# B&R Automation Studio project acopos6d_issues (part 4)

#### PackMLModuleStateManaging.cpp
```cpp
#include "PackMLModule.hpp"

		// -----------------------------------------------------------------------------

const char *internalInfoStateNames[] = { "Undefined",
	"Clearing",
	"Stopped",
	"Starting",
	"Idle",
	"Suspended",
	"Execute",
	"Stopping",
	"Aborting",
	"Aborted",
	"Holding",
	"Held",
	"Unholding",
	"Suspending",
	"Unsuspending",
	"Resetting",
	"Completing",
	"Completed",
	"",
	"",
	"",
	"",
	"",
	"",
	"",
	"",
	"",
	"",
	"",
	"",
	"Deactivating",
	"Deactivated",
	"Activating" };

const char *internalInfoModeNames[] = { "Undefined",
	"Production",
	"Maintenance",
	"Manual",
	""};

		// -----------------------------------------------------------------------------
		// we need to add complete cmd to the pattern
const unsigned long CMD_VALID_BIT_PATTERN_LIST[]
	= { 0,          0x00000080, 0x20004080, 0x000000C0, 0x000000C4, 0x0000A2C0,
	0x000092C0, 0x00000080, 0,          0x20000001, 0x000000C0, 0x000088C0,
	0x000000C0, 0x000000C0, 0x000000C0, 0x000000C0, 0x000000C0, 0x000040C0,
	0,          0,          0,          0,          0,          0,
	0,          0,          0,          0,          0,          0,
	0,          0x80000000, 0 };

// -----------------------------------------------------------------------------

PackMLModule* PackMLModule::getParentPtr(){
	if (!hasParent_)
		return nullptr;

	return pParentLink_;
}
// -----------------------------------------------------------------------------
PackMLModule* PackMLModule::getChildPtr(unsigned long int childIdx){
	if(childCount_ <= 0)
		return nullptr;

	return childLinks_[childIdx % childCount_];
}
// -----------------------------------------------------------------------------
PackMLModule* PackMLModule::getSiblingPtr(unsigned long int siblingIdx){
	if (!hasParent_)
		return nullptr;

	return pParentLink_->getChildPtr(siblingIdx);
}
// -----------------------------------------------------------------------------

PackMLModuleStateEnu PackMLModule::getChildCurrentState(unsigned long int childIndex){
	if(childCount_ <= 0)
		return ST_UNDEFINED;

	return childLinks_[childIndex % childCount_]->getCurrentState();
}
		// -----------------------------------------------------------------------------
long int PackMLModule::getChildCurrentSubState(unsigned long int childIndex){
	if(childCount_ <= 0)
		return 0;

	return childLinks_[childIndex % childCount_]->getCurrentSubState();
}
		// -----------------------------------------------------------------------------
bool PackMLModule::getChildStateComplete(unsigned long int childIndex){
	if(childCount_ <= 0)
		return false;

	return childLinks_[childIndex % childCount_]->getStateComplete();
}
		// -----------------------------------------------------------------------------
const char* PackMLModule::getChildName(unsigned long int childIndex){
	if(childCount_ <= 0)
		return "";

	return childLinks_[childIndex % childCount_]->getModuleName();
}
		// -----------------------------------------------------------------------------
PackMLModuleStateEnu PackMLModule::getSiblingCurrentState(unsigned long int siblingIndex){
	if (!hasParent_)
		return ST_UNDEFINED;

	return pParentLink_->getChildCurrentState(siblingIndex);
}
		// -----------------------------------------------------------------------------
long int PackMLModule::getSiblingCurrentSubState(unsigned long int siblingIndex){
	if (!hasParent_)
		return 0;

	return pParentLink_->getChildCurrentSubState(siblingIndex);
}
		// -----------------------------------------------------------------------------
bool PackMLModule::getSiblingStateComplete(unsigned long int siblingIndex){
	if (!hasParent_)
		return false;

	return pParentLink_->getChildStateComplete(siblingIndex);
}
		// -----------------------------------------------------------------------------
const char* PackMLModule::getSiblingName(unsigned long int siblingIndex){
	if (!hasParent_)
		return "";

	return pParentLink_->getChildName(siblingIndex);
}
		// -----------------------------------------------------------------------------
bool PackMLModule::isChild_(PackMLModule* pModule){
	for (unsigned short i = 0; i < childCount_; ++i) {
		if (childLinks_[i] == pModule) {
			return true;
		}
	}
	return false;
}
		// -----------------------------------------------------------------------------
unsigned long PackMLModule::getSiblingCount(){
	if (!hasParent_) {
		return 1;
	}
	return pParentLink_->getChildCount();
}
		// -----------------------------------------------------------------------------
bool PackMLModule::getSiblingsStateComplete(){
	if (!hasParent_) {
		return stateComplete_;
	}
	return pParentLink_->getChildrenStateComplete();
}

		// -----------------------------------------------------------------------------
bool PackMLModule::getChildrenStateComplete(){
	for (unsigned short i = 0; i < childCount_; ++i) {
		if (!childLinks_[i]->getStateComplete()) {
			return false;
		}
	}
	return true;
}
		// -----------------------------------------------------------------------------
PackMLModuleStateEnu PackMLModule::getParentCurrentState()
{
	if (!hasParent_) {
		return ST_UNDEFINED;
	}
	return pParentLink_->getCurrentState();
}

		// -----------------------------------------------------------------------------

long int PackMLModule::getParentCurrentSubState()
{
	if (!hasParent_) {
		return 0;
	}
	return pParentLink_->getCurrentSubState();
}

		// -----------------------------------------------------------------------------

const char *PackMLModule::getParentName()
{
	if (!hasParent_) {
		return "";
	}
	return pParentLink_->getModuleName();
}

bool PackMLModule::getParentStateComplete()
{
	if (!hasParent_) {
		return true;
	}
	return pParentLink_->getStateComplete();
}

		// -----------------------------------------------------------------------------

const char *PackMLModule::getCurrentStateStr() const
{
	return internalInfoStateNames[stateCurrent_];

}

const char *PackMLModule::getStateStr(PackMLModuleStateEnu state) const
{
	return internalInfoStateNames[state];
}

		// -----------------------------------------------------------------------------

		// -----------------------------------------------------------------------------

const char* PackMLModule::getCurrentModeName() const
{
	return internalInfoModeNames[modeCurrent_];
}

const char* PackMLModule::getModeName(signed long int modeId) const
{
	return internalInfoModeNames[modeId];
}

		// -----------------------------------------------------------------------------

// --------------------------------------------------------------------------

void PackMLModule::setNewModeCurrent(long int mode)
{
	modeCurrent_ = mode;

	for (unsigned short i = 0; i < childCount_; ++i) {
		childLinks_[i]->setNewModeCurrent(modeCurrent_);
	}
}

		// -----------------------------------------------------------------------------

bool PackMLModule::setCurrentMode(long int mode)
{

	// Check if the hierarchy is in synch
	if(!isModeChangePossible())
		return false;

	// update mode
	setNewModeCurrent(mode);
	// propagate mode to the children within one cycle
	return true;
}

		// -----------------------------------------------------------------------------

bool PackMLModule::isModeChangePossible()
{
	// What should the child do when it is not synchronised with the parent?
	if (!childrenInState_(stateCurrent_)) {
		return false;
	}

	for (unsigned short i = 0; i < childCount_; ++i) {
		if (!childLinks_[i]->isModeChangePossible()) {
			return false;
		}
	}

	return true;
}
		// -----------------------------------------------------------------------------

bool PackMLModule::childrenInState_(PackMLModuleStateEnu state)
{

	for (unsigned short i = 0; i < childCount_; ++i) {
		PackMLModuleStateEnu childState = childLinks_[i]->getCurrentState();
		if (childState != state && childState != ST_DEACTIVATED) {
			return false;
		}
	}
	return true;
}

		// -------------------------------------------------------------------------

bool PackMLModule::stateExistInPattern_(unsigned long stateBitPattern,
	PackMLModuleStateEnu state)
{
	if (state == ST_UNDEFINED) {
		return true;
	}
	unsigned long patternChecker = 1;
	return (stateBitPattern & (patternChecker << (state - 1)));
}

		// -------------------------------------------------------------------------

bool PackMLModule::cmdValid_(PackMLModuleStateEnu state)
{

	return stateExistInPattern_(CMD_VALID_BIT_PATTERN_LIST[stateCurrent_],
		state);
}

		// ------------------------------------------------------------------------

bool PackMLModule::isActingState(PackMLModuleStateEnu state)
{
	unsigned long actingStateBitPattern = 0xA000FAC5;

	return stateExistInPattern_(actingStateBitPattern, state);
}

		// -----------------------------------------------------------------------------

// from waiting state to acting state
void PackMLModule::executeCmd_(PackMLModuleStateEnu targetState)
{
	stateCurrent_ = targetState;
	// reset internal bools
	resetInternalCmds_();
	resetWaitingFor_();
	resetInteruptedBy_();
}

		// -----------------------------------------------------------------------------
// from acting state to waiting state
void PackMLModule::executeActingState_(PackMLModuleStateEnu targetState)
{
	if (childrenInSynch_(targetState)) {
		// Update the state
		stateCurrent_ = targetState;
		// reset internal bools
		resetInternalCmds_();
		resetWaitingFor_();
	}
}

		// -----------------------------------------------------------------------------
		// Checks if the children are in the desired state in case where they want to be
		// synchronised
bool PackMLModule::childrenInSynch_(PackMLModuleStateEnu targetState)
{

	for (unsigned long i = 0; i < childCount_; ++i) {
		if ((childLinks_[i]->getCurrentState() != targetState) && childLinks_[i]->needParentSynch(stateCurrent_)) {
			return false;
		}
	}
	return true;
}

		// -----------------------------------------------------------------------------

void PackMLModule::resetInternalCmds_()
{
	if(isActingState(stateCurrent_)){
		externalAbort_ = false;
		externalClear_ = false;
		externalStop_ = false;
		externalReset_ = false;
		externalStart_ = false;
		externalHold_ = false;
		externalUnhold_ = false;
		externalSuspend_ = false;
		externalUnsuspend_ = false;
		externalComplete_ = false;
		externalStateComplete_ = false;
	}

	activate_ = false;
	deactivate_ = false;

	abort_ = externalAbort_;
	clear_ = externalClear_;
	stop_ = externalStop_;
	reset_ = externalReset_;
	start_ = externalStart_;
	hold_ = externalHold_;
	unhold_ = externalUnhold_;
	suspend_ = externalSuspend_;
	unsuspend_ = externalUnsuspend_;
	complete_ = externalComplete_;
	stateComplete_ = false;

	oldAbort_ = false;
	oldClear_ = false;
	oldStop_ = false;
	oldReset_ = false;
	oldStart_ = false;
	oldHold_ = false;
	oldUnhold_ = false;
	oldSuspend_ = false;
	oldUnsuspend_ = false;
	oldComplete_ = false;
	oldStateComplete_ = false;

	timeInState_ = 0.0;
}

		// -----------------------------------------------------------------------------

void PackMLModule::escalateCmdAbort()
{
	if (escalateAbort_) {
		return pParentLink_->escalateCmdAbort();
	}
	abort_ = !overrideAbort_;
	externalAbort_ = abort_;
}
void PackMLModule::escalateCmdClear()
{
	if (escalateClear_) {
		return pParentLink_->escalateCmdClear();
	}
	clear_ = !overrideClear_;
	externalClear_ = clear_;
}
void PackMLModule::escalateCmdStop()
{
	if (escalateStop_) {
		return pParentLink_->escalateCmdStop();
	}
	stop_ = !overrideStop_;
	externalStop_ = stop_;
}
void PackMLModule::escalateCmdReset()
{
	if (escalateReset_) {
		return pParentLink_->escalateCmdReset();
	}
	reset_ = !overrideReset_;
	externalReset_ = reset_;
}
void PackMLModule::escalateCmdHold()
{
	if (escalateHold_) {
		return pParentLink_->escalateCmdHold();
	}
	hold_ = !overrideHold_;
	externalHold_ = hold_;
}
void PackMLModule::escalateCmdUnhold()
{
	if (escalateUnhold_) {
		return pParentLink_->escalateCmdUnhold();
	}
	unhold_ = !overrideUnhold_;
	externalUnhold_ = unhold_;
}
void PackMLModule::escalateCmdSuspend()
{
	if (escalateSuspend_) {
		return pParentLink_->escalateCmdSuspend();
	}
	suspend_ = !overrideSuspend_;
	externalSuspend_ = suspend_;
}
void PackMLModule::escalateCmdUnsuspend()
{
	if (escalateUnsuspend_) {
		return pParentLink_->escalateCmdUnsuspend();
	}
	unsuspend_ = !overrideUnsuspend_;
	externalUnsuspend_ = unsuspend_;
}
void PackMLModule::escalateCmdStart()
{
	if (escalateStart_) {
		return pParentLink_->escalateCmdStart();
	}
	start_ = !overrideStart_;
	externalStart_ = start_;
}
void PackMLModule::escalateCmdComplete()
{
	if (escalateComplete_) {
		return pParentLink_->escalateCmdComplete();
	}
	complete_ = !overrideComplete_;
	externalComplete_ = complete_;
}

// ----------------------------------------------------------------------------

void PackMLModule::propagateCmdAbort(bool root)
{
	abort_ = reactToAbort_ && !root;
	externalAbort_ = abort_;

	for (unsigned short i = 0; i < childCount_; ++i) {
		childLinks_[i]->propagateCmdAbort(false);
	}
}
void PackMLModule::propagateCmdClear(bool root)
{
	clear_ = reactToClear_ && !root;
	externalClear_ = clear_;

	for (unsigned short i = 0; i < childCount_; ++i) {
		childLinks_[i]->propagateCmdClear(false);
	}
}
void PackMLModule::propagateCmdStop(bool root)
{
	stop_ = reactToStop_ && !root;
	externalStop_ = stop_;

	for (unsigned short i = 0; i < childCount_; ++i) {
		childLinks_[i]->propagateCmdStop(false);
	}
}
void PackMLModule::propagateCmdReset(bool root)
{
	reset_ = reactToReset_ && !root;
	externalReset_ = reset_;

	for (unsigned short i = 0; i < childCount_; ++i) {
		childLinks_[i]->propagateCmdReset(false);
	}
}
void PackMLModule::propagateCmdHold(bool root)
{
	hold_ = reactToHold_ && !root;
	externalHold_ = hold_;

	for (unsigned short i = 0; i < childCount_; ++i) {
		childLinks_[i]->propagateCmdHold(false);
	}
}
void PackMLModule::propagateCmdUnhold(bool root)
{
	unhold_ = reactToUnhold_ && !root;
	externalUnhold_ = unhold_;

	for (unsigned short i = 0; i < childCount_; ++i) {
		childLinks_[i]->propagateCmdUnhold(false);
	}
}
void PackMLModule::propagateCmdSuspend(bool root)
{
	suspend_ = reactToSuspend_ && !root;
	externalSuspend_ = suspend_;

	for (unsigned short i = 0; i < childCount_; ++i) {
		childLinks_[i]->propagateCmdSuspend(false);
	}
}
void PackMLModule::propagateCmdUnsuspend(bool root)
{
	unsuspend_ = reactToUnsuspend_ && !root;
	externalUnsuspend_ = unsuspend_;

	for (unsigned short i = 0; i < childCount_; ++i) {
		childLinks_[i]->propagateCmdUnsuspend(false);
	}
}
void PackMLModule::propagateCmdStart(bool root)
{
	start_ = reactToStart_ && !root;
	externalStart_ = start_;

	for (unsigned short i = 0; i < childCount_; ++i) {
		childLinks_[i]->propagateCmdStart(false);
	}
}
void PackMLModule::propagateCmdComplete(bool root)
{
	complete_ = reactToComplete_ && !root;
	externalComplete_ = complete_;

	for (unsigned short i = 0; i < childCount_; ++i) {
		childLinks_[i]->propagateCmdComplete(false);
	}
}

// ----------------------------------------------------------------------------

bool PackMLModule::evaluateCmdAbort(bool& newCmd)
{
	if (newCmd && !oldAbort_) {
		oldAbort_ = true;
		return setCmd_(ST_ABORTING);
	}
	else if (!newCmd && oldAbort_) {
		oldAbort_ = false;
		resetCmd_(ST_ABORTING);
	}
	return true;
}
bool PackMLModule::evaluateCmdStop(bool& newCmd)
{
	if (newCmd && !oldStop_) {
		oldStop_ = true;
		return setCmd_(ST_STOPPING);
	}
	else if (!newCmd && oldStop_) {
		oldStop_ = false;
		resetCmd_(ST_STOPPING);
	}
	return true;
}
bool PackMLModule::evaluateCmdClear(bool& newCmd)
{
	if (newCmd && !oldClear_) {
		oldClear_ = true;
		return setCmd_(ST_CLEARING);
	}
	else if (!newCmd && oldClear_) {
		oldClear_ = false;
		resetCmd_(ST_CLEARING);
	}
	return true;
}
bool PackMLModule::evaluateCmdReset(bool& newCmd)
{
	if (newCmd && !oldReset_) {
		oldReset_ = true;
		return setCmd_(ST_RESETTING);
	}
	else if (!newCmd && oldReset_) {
		oldReset_ = false;
		resetCmd_(ST_RESETTING);
	}
	return true;
}
bool PackMLModule::evaluateCmdStart(bool& newCmd)
{
	if (newCmd && !oldStart_) {
		oldStart_ = true;
		return setCmd_(ST_STARTING);
	}
	else if (!newCmd && oldStart_) {
		oldStart_ = false;
		resetCmd_(ST_STARTING);
	}
	return true;
}
bool PackMLModule::evaluateCmdSuspend(bool& newCmd)
{
	if (newCmd && !oldSuspend_) {
		oldSuspend_ = true;
		return setCmd_(ST_SUSPENDING);
	}
	else if (!newCmd && oldSuspend_) {
		oldSuspend_ = false;
		resetCmd_(ST_SUSPENDING);
	}
	return true;
}
bool PackMLModule::evaluateCmdUnsuspend(bool& newCmd)
{
	if (newCmd && !oldUnsuspend_) {
		oldUnsuspend_ = true;
		return setCmd_(ST_UNSUSPENDING);
	}
	else if (!newCmd && oldUnsuspend_) {
		oldUnsuspend_ = false;
		resetCmd_(ST_UNSUSPENDING);
	}
	return true;
}
bool PackMLModule::evaluateCmdHold(bool& newCmd)
{
	if (newCmd && !oldHold_) {
		oldHold_ = true;
		return setCmd_(ST_HOLDING);
	}
	else if (!newCmd && oldHold_) {
		oldHold_ = false;
		resetCmd_(ST_HOLDING);
	}
	return true;
}
bool PackMLModule::evaluateCmdUnhold(bool& newCmd)
{
	if (newCmd && !oldUnhold_) {
		oldUnhold_ = true;
		return setCmd_(ST_UNHOLDING);
	}
	else if (!newCmd && oldUnhold_) {
		oldUnhold_ = false;
		resetCmd_(ST_UNHOLDING);
	}
	return true;
}
bool PackMLModule::evaluateCmdComplete(bool& newCmd)
{
	if (newCmd && !oldComplete_) {
		oldComplete_ = true;
		return setCmd_(ST_COMPLETING);
	}
	else if (!newCmd && oldComplete_) {
		oldComplete_ = false;
		resetCmd_(ST_COMPLETING);
	}
	return true;
}
bool PackMLModule::evaluateCmdStateComplete(bool& newCmd)
{
	if (newCmd && !oldStateComplete_) {
		oldStateComplete_ = true;
		return setCmd_(ST_UNDEFINED);
	}
	else if (!newCmd && oldStateComplete_) {
		oldStateComplete_ = false;
		resetCmd_(ST_UNDEFINED);
	}
	return true;
}

bool PackMLModule::setCmdAbort(){
	return setCmd_(ST_ABORTING);
}
bool PackMLModule::setCmdStop(){
	return setCmd_(ST_STOPPING);
}
bool PackMLModule::setCmdClear(){
	return setCmd_(ST_CLEARING);
}
bool PackMLModule::setCmdReset(){
	return setCmd_(ST_RESETTING);
}
bool PackMLModule::setCmdStart(){
	return setCmd_(ST_STARTING);
}
bool PackMLModule::setCmdSuspend(){
	return setCmd_(ST_SUSPENDING);
}
bool PackMLModule::setCmdUnsuspend(){
	return setCmd_(ST_UNSUSPENDING);
}
bool PackMLModule::setCmdHold(){
	return setCmd_(ST_HOLDING);
}
bool PackMLModule::setCmdUnhold(){
	return setCmd_(ST_UNHOLDING);
}
bool PackMLModule::setCmdComplete(){
	return setCmd_(ST_COMPLETING);
}
bool PackMLModule::setCmdStateComplete(){
	return setCmd_(ST_UNDEFINED);
}

void PackMLModule::resetCmdAbort(){
	return resetCmd_(ST_ABORTING);
}
void PackMLModule::resetCmdStop(){
	return resetCmd_(ST_STOPPING);
}
void PackMLModule::resetCmdClear(){
	return resetCmd_(ST_CLEARING);
}
void PackMLModule::resetCmdReset(){
	return resetCmd_(ST_RESETTING);
}
void PackMLModule::resetCmdStart(){
	return resetCmd_(ST_STARTING);
}
void PackMLModule::resetCmdSuspend(){
	return resetCmd_(ST_SUSPENDING);
}
void PackMLModule::resetCmdUnsuspend(){
	return resetCmd_(ST_UNSUSPENDING);
}
void PackMLModule::resetCmdHold(){
	return resetCmd_(ST_HOLDING);
}
void PackMLModule::resetCmdUnhold(){
	return resetCmd_(ST_UNHOLDING);
}
void PackMLModule::resetCmdComplete(){
	return resetCmd_(ST_COMPLETING);
}
void PackMLModule::resetCmdStateComplete(){
	return resetCmd_(ST_UNDEFINED);
}

		// -----------------------------------------------------------------------------

bool PackMLModule::setCmd_(PackMLModuleStateEnu targetActingState) // NOLINT
{

	bool cmdValid = cmdValid_(targetActingState);

	switch (targetActingState) { // NOCCM
		case ST_CLEARING:
			if (overrideClear_ && !escalateClear_) {
				return false; // error code
			}
			if (hasParent_ && escalateClear_ && cmdValid) {
				pParentLink_->escalateCmdClear();
				setInteruptedBy_();
			}
			clear_ = !overrideClear_; //!overrideAbort_ || !escalateAbort_;
			break;

		case ST_STARTING:
			if (overrideStart_ && !escalateStart_) {
				return false; // error code
			}
			if (hasParent_ && escalateStart_ && cmdValid) {
				pParentLink_->escalateCmdStart();
				setInteruptedBy_();
			}
			start_ = !overrideStart_;
			break;

		case ST_STOPPING:
			if (overrideStop_ && !escalateStop_) {
				return false; // error code
			}
			if (hasParent_ && escalateStop_) {
				pParentLink_->escalateCmdStop();
			}
			if(cmdValid){
				setInteruptedBy_();
				stop_ = !overrideStop_;
			}
			break;

		case ST_ABORTING:
			if (overrideAbort_ && !escalateAbort_) {
				return false; // error code
			}
			if (hasParent_ && escalateAbort_) {
				pParentLink_->escalateCmdAbort();
			}

			if(cmdValid){
				setInteruptedBy_();
				abort_ = !overrideAbort_;
			}
			break;

		case ST_HOLDING:
			if (overrideHold_ && !escalateHold_) {
				return false; // error code
			}
			if (hasParent_ && escalateHold_) {
				pParentLink_->escalateCmdHold();
			}
			if(cmdValid){
				setInteruptedBy_();
				hold_ = !overrideHold_;
			}
			break;

		case ST_UNHOLDING:
			if (overrideUnhold_ && !escalateUnhold_) {
				return false; // error code
			}
			if (hasParent_ && escalateUnhold_ && cmdValid) {
				pParentLink_->escalateCmdUnhold();
				setInteruptedBy_();
			}
			unhold_ = !overrideUnhold_;
			break;

		case ST_SUSPENDING:
			if (overrideSuspend_ && !escalateSuspend_) {
				return false; // error code
			}
			if (hasParent_ && escalateSuspend_) {
				pParentLink_->escalateCmdSuspend();
			}
			if(cmdValid){
				setInteruptedBy_();
				suspend_ = !overrideSuspend_;
			}
			break;

		case ST_UNSUSPENDING:
			if (overrideUnsuspend_ && !escalateUnsuspend_) {
				return false; // error code
			}
			if (hasParent_ && escalateUnsuspend_ && cmdValid) {
				pParentLink_->escalateCmdUnsuspend();
				setInteruptedBy_();
			}
			unsuspend_ = !overrideUnsuspend_;
			break;

		case ST_RESETTING:
			if (overrideReset_ && !escalateReset_) {
				return false; // error code
			}
			if (hasParent_ && escalateReset_ && cmdValid) {
				pParentLink_->escalateCmdReset();
				setInteruptedBy_();
			}
			reset_ = !overrideReset_;
			break;

		case ST_COMPLETING:
			// check if the state group is configured
			if (overrideComplete_ && !escalateComplete_) {
				return false; // error code
			}
			if (hasParent_ && escalateComplete_) {
				pParentLink_->escalateCmdComplete();
			}
			if(cmdValid){
				setInteruptedBy_();
				complete_ = !overrideComplete_;
			}
			break;

		case ST_UNDEFINED:
			stateComplete_ = true;
			break;

		default:
			break;
	}

	return true;
}

		// -----------------------------------------------------------------------------

void PackMLModule::resetCmd_(PackMLModuleStateEnu targetActingState)
{

	switch (targetActingState) { // NOCCM
		case ST_CLEARING:
			clear_ = externalClear_;
			break;

		case ST_STARTING:
			start_ = externalStart_;
			break;

		case ST_STOPPING:
			stop_ = externalStop_;
			break;

		case ST_ABORTING:
			abort_ = externalAbort_;
			break;

		case ST_HOLDING:
			hold_ = externalHold_;
			break;

		case ST_UNHOLDING:
			unhold_ = externalUnhold_;
			break;

		case ST_SUSPENDING:
			suspend_ = externalSuspend_;
			break;

		case ST_UNSUSPENDING:
			unsuspend_ = externalUnsuspend_;
			break;

		case ST_RESETTING:
			reset_ = externalReset_;
			break;

		case ST_COMPLETING:
			complete_ = externalComplete_;
			break;

		case ST_UNDEFINED:
			stateComplete_ = externalStateComplete_;
			break;

		default:
			break;
	}
}

		// -----------------------------------------------------------------------------

		// if parent synchronisation needed
bool PackMLModule::needParentSynch(PackMLModuleStateEnu state)
{
	if (hierarchyLevel_ == 0) {
		return true;
	}

	switch (stateCurrent_) { // NOCCM

		case ST_CLEARING:
			switch (state) { // NOCCM
				case ST_ABORTING:
					return overrideAbort_ || reactToAbort_;
				case ST_CLEARING:
					return overrideClear_ || reactToClear_;
				default:
					break;
			}
			break;

		case ST_STOPPED:
			switch (state) { // NOCCM
				case ST_ABORTING:
					return overrideAbort_ || reactToAbort_;
				case ST_RESETTING:
					return overrideReset_ || reactToReset_;
				default:
					break;
			}
			break;

		case ST_IDLE:
			switch (state) { // NOCCM
				case ST_ABORTING:
					return overrideAbort_ || reactToAbort_;
				case ST_STOPPING:
					return overrideStop_ || reactToStop_;
				case ST_STARTING:
					return overrideStart_ || reactToStart_;
				default:
					break;
			}
			break;

		case ST_SUSPENDED:
			switch (state) { // NOCCM
				case ST_ABORTING:
					return overrideAbort_ || reactToAbort_;
				case ST_STOPPING:
					return overrideStop_ || reactToStop_;
				case ST_UNSUSPENDING:
					return overrideUnsuspend_ || reactToUnsuspend_;
				case ST_HOLDING:
					return overrideHold_ || reactToHold_;
				case ST_COMPLETING:
					return overrideComplete_ || reactToComplete_;
				default:
					break;
			}
			break;

		case ST_EXECUTE:
			switch (state) { // NOCCM
				case ST_ABORTING:
					return overrideAbort_ || reactToAbort_;
				case ST_STOPPING:
					return overrideStop_ || reactToStop_;
				case ST_SUSPENDING:
					return overrideSuspend_ || reactToSuspend_;
				case ST_HOLDING:
					return overrideHold_ || reactToHold_;
				case ST_COMPLETING:
					return overrideComplete_ || reactToComplete_;
				default:
					break;
			}
			break;

		case ST_STOPPING:
			switch (state) { // NOCCM
				case ST_ABORTING:
					return overrideAbort_ || reactToAbort_;
				case ST_STOPPING:
					return overrideStop_ || reactToStop_;
				default:
					break;
			}
			break;

		case ST_ABORTING:
			switch (state) { // NOCCM
				case ST_ABORTING:
					return overrideAbort_ || reactToAbort_;
				default:
					break;
			}
			break;

		case ST_ABORTED:
			switch (state) { // NOCCM
				case ST_CLEARING:
					return overrideClear_ || reactToClear_;
				default:
					break;
			}
			break;

		case ST_HELD:
			switch (state) { // NOCCM
				case ST_ABORTING:
					return overrideAbort_ || reactToAbort_;
				case ST_STOPPING:
					return overrideStop_ || reactToStop_;
				case ST_UNHOLDING:
					return overrideUnhold_ || reactToUnhold_;
				case ST_COMPLETING:
					return overrideComplete_ || reactToComplete_;
				default:
					break;
			}
			break;

		case ST_SUSPENDING:
			switch (state) { // NOCCM
				case ST_ABORTING:
					return overrideAbort_ || reactToAbort_;
				case ST_STOPPING:
					return overrideStop_ || reactToStop_;
				case ST_SUSPENDING:
					return overrideSuspend_ || reactToSuspend_;
				default:
					break;
			}
			break;
		case ST_UNSUSPENDING:
			switch (state) { // NOCCM
				case ST_ABORTING:
					return overrideAbort_ || reactToAbort_;
				case ST_STOPPING:
					return overrideStop_ || reactToStop_;
				case ST_UNSUSPENDING:
					return overrideUnsuspend_ || reactToUnsuspend_;
				default:
					break;
			}
			break;
		case ST_COMPLETING:
			switch (state) { // NOCCM
				case ST_ABORTING:
					return overrideAbort_ || reactToAbort_;
				case ST_STOPPING:
					return overrideStop_ || reactToStop_;
				case ST_COMPLETING:
					return overrideComplete_ || reactToComplete_;
				default:
					break;
			}
			break;
		case ST_STARTING:
			switch (state) { // NOCCM
				case ST_ABORTING:
					return overrideAbort_ || reactToAbort_;
				case ST_STOPPING:
					return overrideStop_ || reactToStop_;
				case ST_STARTING:
					return overrideStart_ || reactToStart_;
				default:
					break;
			}
			break;
		case ST_HOLDING:
			switch (state) { // NOCCM
				case ST_ABORTING:
					return overrideAbort_ || reactToAbort_;
				case ST_STOPPING:
					return overrideStop_ || reactToStop_;
				case ST_HOLDING:
					return overrideHold_ || reactToHold_;
				default:
					break;
			}
			break;
		case ST_UNHOLDING:
			switch (state) { // NOCCM
				case ST_ABORTING:
					return overrideAbort_ || reactToAbort_;
				case ST_STOPPING:
					return overrideStop_ || reactToStop_;
				case ST_UNHOLDING:
					return overrideUnhold_ || reactToUnhold_;
				default:
					break;
			}
			break;

		case ST_RESETTING:
			switch (state) { // NOCCM
				case ST_ABORTING:
					return overrideAbort_ || reactToAbort_;
				case ST_STOPPING:
					return overrideStop_ || reactToStop_;
				case ST_RESETTING:
					return overrideReset_ || reactToReset_;
				default:
					break;
			}
			break;

		case ST_COMPLETE:
			switch (state) { // NOCCM
				case ST_ABORTING:
					return overrideAbort_ || reactToAbort_;
				case ST_STOPPING:
					return overrideStop_ || reactToStop_;
				case ST_RESETTING:
					return overrideReset_ || reactToReset_;
				default:
					break;
			}
			break;

		default:
			break;
	}

	return false;
}

// -----------------------------------------------------------------------------
// decide if reacto to only should when parent + 1 state in front of child. e.g. instead of ST_ABORTING and ST_ABORTED --> only ST_ABORTING
void PackMLModule::checkParentStateCondition_()
{
	if (hierarchyLevel_ == 0) {
		return;
	}

	PackMLModuleStateEnu parentState = getParentCurrentState();

	if (parentState == stateCurrent_) {
		return;
	}

	switch (stateCurrent_) { // NOCCM
		case ST_CLEARING:
			switch (parentState) { // NOCCM
				case ST_ABORTING:
					abort_ = overrideAbort_ || abort_ || reactToAbort_;
					break;
				case ST_ABORTED:
					abort_ = overrideAbort_ || abort_;
					break;
				default:
					break;
			}
			break;

		case ST_STOPPED:
			switch (parentState) { // NOCCM
				case ST_ABORTING:
					abort_ = overrideAbort_ || abort_ || reactToAbort_;
					break;
				case ST_ABORTED:
					abort_ = overrideAbort_ || abort_;
					break;

				case ST_DEACTIVATING:
				case ST_DEACTIVATED:
					deactivate_ = (activationCondition_ == 1);
					break;

				case ST_RESETTING:
					reset_ = overrideReset_ || reset_ || reactToReset_;
					break;

				case ST_IDLE:
				case ST_STARTING:
				case ST_SUSPENDED:
				case ST_EXECUTE:
				case ST_HOLDING:
				case ST_HELD:
				case ST_UNHOLDING:
				case ST_SUSPENDING:
				case ST_UNSUSPENDING:
				case ST_COMPLETING:
				case ST_COMPLETE:
					reset_ = overrideReset_ || reset_;
					break;

				default:
					break;
			}
			break;

		case ST_IDLE:
			switch (parentState) { // NOCCM
				case ST_ABORTING:
					abort_ = overrideAbort_ || abort_ || reactToAbort_;
					break;
				case ST_ABORTED:
					abort_ = overrideAbort_ || abort_;
					break;

				case ST_CLEARING:
					stop_ = overrideStop_ || stop_;
					abort_ = (overrideAbort_ || abort_) && !stop_;
					break;

				case ST_STOPPING:
					stop_ = overrideStop_ || stop_ || reactToStop_;
					break;
				case ST_STOPPED:
					stop_ = overrideStop_ || stop_;
					break;

				case ST_DEACTIVATING:
				case ST_DEACTIVATED:
				case ST_ACTIVATING:
					stop_ = overrideStop_ || stop_;
					abort_ = (overrideAbort_ || abort_) && !stop_;
					break;

				case ST_STARTING:
					start_ = overrideStart_ || start_ || reactToStart_;
					break;

				case ST_EXECUTE:
				case ST_SUSPENDED:
				case ST_HOLDING:
				case ST_HELD:
				case ST_UNHOLDING:
				case ST_SUSPENDING:
				case ST_UNSUSPENDING:
				case ST_COMPLETING:
				case ST_COMPLETE:
					start_ = overrideStart_ || start_;
					break;

				default:
					break;
			}
			break;

		case ST_SUSPENDED:
			switch (parentState) { // NOCCM
				case ST_ABORTING:
					abort_ = overrideAbort_ || abort_ || reactToAbort_;
					break;
				case ST_ABORTED:
					abort_ = overrideAbort_ || abort_;
					break;

				case ST_CLEARING:
					stop_ = overrideStop_ || stop_;
					abort_ = (overrideAbort_ || abort_) && !stop_;
					break;

				case ST_STOPPING:
					stop_ = overrideStop_ || stop_ || reactToStop_;
					break;
				case ST_STOPPED:
					stop_ = overrideStop_ || stop_;
					break;

				case ST_UNSUSPENDING:
					unsuspend_ = overrideUnsuspend_ || unsuspend_ || reactToUnsuspend_;
					break;

				case ST_DEACTIVATING:
				case ST_DEACTIVATED:
				case ST_ACTIVATING:
					stop_ = overrideStop_ || stop_;
					abort_ = (overrideAbort_ || abort_) && !stop_;
					break;

				case ST_RESETTING:
				case ST_IDLE: // **********************
					unsuspend_ = overrideUnsuspend_ || unsuspend_;
					stop_ = (overrideStop_ || stop_) && !unsuspend_;
					break;

				case ST_COMPLETING:
					complete_ = overrideComplete_ || complete_ || reactToComplete_;
					break;
				case ST_COMPLETE:
					complete_ = overrideComplete_ || complete_;
					break;

				case ST_HOLDING:
					hold_ = overrideHold_ || hold_ || reactToHold_;
					break;
				case ST_HELD:
					hold_ = overrideHold_ || hold_;
					break;

				case ST_EXECUTE:
				case ST_STARTING:
				case ST_UNHOLDING:
					unsuspend_ = overrideUnsuspend_ || unsuspend_;
					break;

				default:
					break;
			}
			break;

		case ST_EXECUTE:
			switch (parentState) { // NOCCM
				case ST_ABORTING:
					abort_ = overrideAbort_ || abort_ || reactToAbort_;
					break;
				case ST_ABORTED:
					abort_ = overrideAbort_ || abort_;
					break;

				case ST_CLEARING:
					stop_ = overrideStop_ || stop_;
					abort_ = (overrideAbort_ || abort_) && !stop_;
					break;

				case ST_STOPPING:
					stop_ = overrideStop_ || stop_ || reactToStop_;
					break;

				case ST_STOPPED:
					stop_ = overrideStop_ || stop_;
					break;

				case ST_SUSPENDING:
					suspend_ = overrideSuspend_ || suspend_ || reactToSuspend_;
					break;

				case ST_SUSPENDED:
					suspend_ = overrideSuspend_ || suspend_;
					break;

				case ST_HOLDING:
					hold_ = overrideHold_ || hold_ || reactToHold_;
					break;

				case ST_HELD:
					hold_ = overrideHold_ || hold_;
					break;

				case ST_COMPLETING:
					complete_ = overrideComplete_ || complete_ || reactToComplete_;
					break;

				case ST_COMPLETE:
					complete_ = overrideComplete_ || complete_;
					break;

				case ST_DEACTIVATING:
				case ST_DEACTIVATED:
				case ST_ACTIVATING:
					stop_ = overrideStop_ || stop_;
					abort_ = (overrideAbort_ || abort_) && !stop_;
					break;

				case ST_RESETTING:
				case ST_IDLE:
					complete_ = overrideComplete_ || complete_;
					stop_ = (overrideStop_ || stop_) && !complete_;
					break;

				default:
					break;
			}
			break;

		case ST_STOPPING:
			switch (parentState) { // NOCCM
				case ST_ABORTING:
					abort_ = overrideAbort_ || abort_ || reactToAbort_;
					break;
				case ST_ABORTED:
					abort_ = overrideAbort_ || abort_;
					break;
				default:
					break;
			}
			break;

		case ST_ABORTED:
			switch (parentState) { // NOCCM
				case ST_DEACTIVATING:
				case ST_DEACTIVATED:
					deactivate_ = (activationCondition_ == 1);
					break;

				case ST_CLEARING:
					clear_ = overrideClear_ || clear_ || reactToClear_;
					break;

				case ST_STOPPED:
				case ST_STARTING:
				case ST_IDLE:
				case ST_SUSPENDED:
				case ST_EXECUTE:
				case ST_STOPPING:
				case ST_HOLDING:
				case ST_HELD:
				case ST_UNHOLDING:
				case ST_SUSPENDING:
				case ST_UNSUSPENDING:
				case ST_RESETTING:
				case ST_COMPLETING:
				case ST_COMPLETE:
				case ST_ACTIVATING:
					clear_ = overrideClear_ || clear_;
					break;

				default:
					break;
			}
			break;

		case ST_HELD:
			switch (parentState) { // NOCCM
				case ST_ABORTING:
					abort_ = overrideAbort_ || abort_ || reactToAbort_;
					break;
				case ST_ABORTED:
					abort_ = overrideAbort_ || abort_;
					break;

				case ST_CLEARING:
					stop_ = overrideStop_ || stop_;
					abort_ = (overrideAbort_ || abort_) && !stop_;
					break;

				case ST_STOPPING:
					stop_ = overrideStop_ || stop_ || reactToStop_;
					break;

				case ST_STOPPED:
					stop_ = overrideStop_ || stop_;
					break;

				case ST_UNHOLDING:
					unhold_ = overrideUnhold_ || unhold_ || reactToUnhold_;
					break;

				case ST_DEACTIVATING:
				case ST_DEACTIVATED:
				case ST_ACTIVATING:
					stop_ = overrideStop_ || stop_;
					abort_ = (overrideAbort_ || abort_) && !stop_;
					break;

				case ST_RESETTING:
				case ST_IDLE: // **********************
					unhold_ = overrideUnhold_ || unhold_;
					stop_ = (overrideStop_ || stop_) && !unhold_;
					break;

				case ST_COMPLETING:
					complete_ = overrideComplete_ || complete_ || reactToComplete_;
					break;
				case ST_COMPLETE:
					complete_ = overrideComplete_ || complete_;
					break;

				case ST_EXECUTE:
				case ST_SUSPENDING:
				case ST_SUSPENDED:
				case ST_UNSUSPENDING:
				case ST_STARTING:
					unhold_ = overrideUnhold_ || unhold_;
					break;

				default:
					break;
			}
			break;

		case ST_STARTING:
		case ST_HOLDING:
		case ST_UNHOLDING:
		case ST_SUSPENDING:
		case ST_UNSUSPENDING:
			switch (parentState) { // NOCCM
				case ST_ABORTING:
					abort_ = overrideAbort_ || abort_ || reactToAbort_;
					break;

				case ST_ABORTED:
					abort_ = overrideAbort_ || abort_;
					break;

				case ST_CLEARING:
					stop_ = overrideStop_ || stop_;
					abort_ = (overrideAbort_ || abort_) && !stop_;
					break;

				case ST_STOPPING:
					stop_ = overrideStop_ || stop_ || reactToStop_;
					break;

				case ST_STOPPED:
					stop_ = overrideStop_ || stop_;
					break;

				case ST_DEACTIVATING:
				case ST_DEACTIVATED:
				case ST_ACTIVATING:
					stop_ = overrideStop_ || stop_;
					abort_ = (overrideAbort_ || abort_) && !stop_;
					break;

				case ST_RESETTING:
				case ST_IDLE:
					stop_ = overrideStop_ || stop_;
					break;

				default:
					break;
			}
			break;

		case ST_RESETTING:
		case ST_COMPLETING:
			switch (parentState) { // NOCCM
				case ST_ABORTING:
					abort_ = overrideAbort_ || abort_ || reactToAbort_;
					break;
				case ST_ABORTED:
					abort_ = overrideAbort_ || abort_;
					break;

				case ST_CLEARING:
					stop_ = overrideStop_ || stop_;
					abort_ = (overrideAbort_ || abort_) && !stop_;
					break;

				case ST_STOPPING:
					stop_ = overrideStop_ || stop_ || reactToStop_;
					break;

				case ST_STOPPED:
					stop_ = overrideStop_ || stop_;
					break;

				case ST_DEACTIVATING:
				case ST_DEACTIVATED:
				case ST_ACTIVATING:
					stop_ = overrideStop_ || stop_;
					abort_ = (overrideAbort_ || abort_) && !stop_;
					break;

				default:
					break;
			}
			break;

		case ST_COMPLETE:
			switch (parentState) { // NOCCM
				case ST_ABORTING:
					abort_ = overrideAbort_ || abort_ || reactToAbort_;
					break;
				case ST_ABORTED:
					abort_ = overrideAbort_ || abort_;
					break;

				case ST_CLEARING:
					stop_ = overrideStop_ || stop_;
					abort_ = (overrideAbort_ || abort_) && !stop_;
					break;

				case ST_STOPPING:
					stop_ = overrideStop_ || stop_ || reactToStop_;
					break;

				case ST_STOPPED:
					stop_ = overrideStop_ || stop_;
					break;

				case ST_DEACTIVATING:
				case ST_DEACTIVATED:
				case ST_ACTIVATING:
					stop_ = overrideStop_ || stop_;
					abort_ = (overrideAbort_ || abort_) && !stop_;
					break;

				case ST_RESETTING:
					reset_ = overrideReset_ || reset_ || reactToReset_;
					break;

				case ST_IDLE:
				case ST_STARTING:
				case ST_SUSPENDED:
				case ST_EXECUTE:
				case ST_HOLDING:
				case ST_HELD:
				case ST_UNHOLDING:
				case ST_SUSPENDING:
				case ST_UNSUSPENDING:
					reset_ = overrideReset_ || reset_;
					break;

				default:
					break;
			}
			break;

		case ST_DEACTIVATED:
			if (parentState != ST_DEACTIVATING) {
				activate_ = (activationCondition_ == 1);
			}
			break;

		default:
			break;
	}

}

void PackMLModule::resetWaitingFor_()
{
		if(pWaitingFor_ == nullptr)
			return;

	pWaitingFor_->resetValues(moduleId_);
}

void PackMLModule::setWaitingFor_()
{
		if(pWaitingFor_ == nullptr)
			return;

	pWaitingFor_->setValues(moduleName_.c_str(), modeCurrent_, stateCurrent_, subStateCurrent_, stateComplete_, hierarchyLevel_, moduleId_, stateInfo_.c_str());

}

	//	 -----------------------------------------------------------------------------

void PackMLModule::resetInteruptedBy_()
{
	if(pInteruptedBy_ == nullptr)
		return;

	PackMLModuleStateEnu state = pInteruptedBy_->getStateCurrent();
	switch(state){
		case ST_EXECUTE:
			if(stateCurrent_ == ST_ABORTING || stateCurrent_ == ST_SUSPENDING || stateCurrent_ == ST_HOLDING || stateCurrent_ == ST_STOPPING || stateCurrent_ == ST_COMPLETING)
				return;
			break;

		case ST_STOPPED:
			if(stateCurrent_ == ST_ABORTING || stateCurrent_ == ST_RESETTING)
				return;
			break;

		case ST_IDLE:
			if(stateCurrent_ == ST_ABORTING || stateCurrent_ == ST_STOPPING || stateCurrent_ == ST_STARTING)
				return;
			break;

		case ST_HELD:
			if(stateCurrent_ == ST_ABORTING || stateCurrent_ == ST_STOPPING || stateCurrent_ == ST_UNHOLDING)
				return;
			break;

		case ST_SUSPENDED:
			if(stateCurrent_ == ST_ABORTING || stateCurrent_ == ST_STOPPING || stateCurrent_ == ST_UNSUSPENDING)
				return;
			break;

		case ST_ABORTED:
			if(stateCurrent_ == ST_CLEARING)
				return;
			break;

		case ST_COMPLETE:
			if(stateCurrent_ == ST_ABORTING || stateCurrent_ == ST_STOPPING || stateCurrent_ == ST_RESETTING)
				return;
			break;

	//	case ST_RESETTING: ST_STARTING: ST_HOLDING: ST_UNHOLDING: ST_SUSPENDING: ST_UNSUSPENDING: ST_COMPLETING: ST_STOPPING: ST_ABORTING: ST_CLEARING:
		default:
			if(stateCurrent_ == ST_ABORTING || stateCurrent_ == ST_STOPPING)
				return;
			break;

	}

	pInteruptedBy_->resetValues(moduleId_);
}

void PackMLModule::setInteruptedBy_()
{
		if(pInteruptedBy_ == nullptr)
			return;

	pInteruptedBy_->setValues(moduleName_.c_str(), modeCurrent_, stateCurrent_, subStateCurrent_, stateComplete_, pInteruptedBy_->getHierarchyLevel() + 1, moduleId_, stateInfo_.c_str());

}

void PackMLModule::setInteruptedBy(PackMLModule* pPackMLModule)
{
		if(pInteruptedBy_ == nullptr)
			return;

	pInteruptedBy_->setValues(pPackMLModule->moduleName_.c_str(), pPackMLModule->modeCurrent_, pPackMLModule->stateCurrent_, pPackMLModule->subStateCurrent_, pPackMLModule->stateComplete_, pPackMLModule->pInteruptedBy_->getHierarchyLevel() + 1, moduleId_, stateInfo_.c_str());

}

		// -----------------------------------------------------------------------------

void PackMLModule::updatePackMLModel_()
{

	switch (stateCurrent_) { // NOCCM
		case ST_UNDEFINED:
			break;

		case ST_STOPPING:
		case ST_CLEARING:
			if (abort_) {
				executeCmd_(ST_ABORTING);
			}
			else if (stateComplete_) {
				executeActingState_(ST_STOPPED);
			}
			else if (needParentSynch(stateCurrent_)) {
				setWaitingFor_();
			}
			break;

		case ST_STOPPED:
			checkActivationCondition_();
			if (abort_) {
				executeCmd_(ST_ABORTING);
			}
			else if (stateComplete_) {
				if (reset_) {
					executeCmd_(ST_RESETTING);
				}
				else if (deactivate_) {
					executeCmd_(ST_DEACTIVATING);
				}
			}
			else if (reset_ || deactivate_) {
				setWaitingFor_();
			}
			break;

		case ST_IDLE:
			if (abort_) {
				executeCmd_(ST_ABORTING);
			}
			else if (stateComplete_) {
				if (stop_) {
					executeCmd_(ST_STOPPING);
				}
				else if (start_) {
					executeCmd_(ST_STARTING);
				}
			}
			else if (stop_ || start_) {
				setWaitingFor_();
			}
			break;

		case ST_SUSPENDED:
			if (abort_) {
				executeCmd_(ST_ABORTING);
			}
			else if (stateComplete_) {
				if (stop_) {
					executeCmd_(ST_STOPPING);
				}
				else if (complete_) {
					executeCmd_(ST_COMPLETING);
				}
				else if (hold_){
					executeCmd_(ST_HOLDING);
				}
				else if (unsuspend_){
					executeCmd_(ST_UNSUSPENDING);
				}
			}
			else if (stop_ || unsuspend_ || hold_ || complete_) {
				setWaitingFor_();
			}
			break;

		case ST_EXECUTE:
			if (abort_) {
				executeCmd_(ST_ABORTING);
			}
			else if (stateComplete_) {
				if (stop_) {
					executeCmd_(ST_STOPPING);
				}
				else if (complete_) {
					executeCmd_(ST_COMPLETING);
				}
				else if (hold_) {
					executeCmd_(ST_HOLDING);
				}
				else if (suspend_) {
					executeCmd_(ST_SUSPENDING);
				}
			}
			else if (stop_ || suspend_ || hold_ || complete_) {
				setWaitingFor_();
			}
			break;

		case ST_ABORTING:
			if (stateComplete_) {
				executeActingState_(ST_ABORTED);
			}
			else if (needParentSynch(stateCurrent_)) {
				setWaitingFor_();
			}
			break;

		case ST_ABORTED:
			checkActivationCondition_();
			if (stateComplete_) {
				if (clear_) {
					executeCmd_(ST_CLEARING);
				}
				else if (deactivate_) {
					executeCmd_(ST_DEACTIVATING);
				}
			}
			else if (clear_ || deactivate_) {
				setWaitingFor_();
			}
			break;

		case ST_HELD:
			if (abort_) {
				executeCmd_(ST_ABORTING);
			}
			else if (stateComplete_) {
				if (stop_) {
					executeCmd_(ST_STOPPING);
				}
				else if (complete_) {
					executeCmd_(ST_COMPLETING);
				}
				else if (unhold_){
					executeCmd_(ST_UNHOLDING);
				}
			}
			else if (stop_ || unhold_ || complete_) {
				setWaitingFor_();
			}
			break;

		case ST_STARTING:
		case ST_UNHOLDING:
		case ST_UNSUSPENDING:
			if (abort_) {
				executeCmd_(ST_ABORTING);
			}
			else if (stateComplete_) {
				if (stop_) {
					executeCmd_(ST_STOPPING);
				}
				else {
					executeActingState_(ST_EXECUTE);
				}
			}
			else if (needParentSynch(stateCurrent_)) {
				setWaitingFor_();
			}
			break;

		case ST_RESETTING:
			if (abort_) {
				executeCmd_(ST_ABORTING);
			}
			else if (stateComplete_) {
				if (stop_) {
					executeCmd_(ST_STOPPING);
				}
				else {
					executeActingState_(ST_IDLE);
				}
			}
			else if (needParentSynch(stateCurrent_)) {
				setWaitingFor_();
			}
			break;

		case ST_COMPLETING:
			if (abort_) {
				executeCmd_(ST_ABORTING);
			}
			else if (stateComplete_) {
				if (stop_) {
					executeCmd_(ST_STOPPING);
				}
				else {
					executeActingState_(ST_COMPLETE);
				}
			}
			else if (needParentSynch(stateCurrent_)) {
				setWaitingFor_();
			}
			break;

		case ST_HOLDING:
			if (abort_) {
				executeCmd_(ST_ABORTING);
			}
			else if (stateComplete_) {
				if (stop_) {
					executeCmd_(ST_STOPPING);
				}
				else {
					executeActingState_(ST_HELD);
				}
			}
			else if (needParentSynch(stateCurrent_)) {
				setWaitingFor_();
			}
			break;

		case ST_SUSPENDING:
			if (abort_) {
				executeCmd_(ST_ABORTING);
			}
			else if (stateComplete_) {
				if (stop_) {
					executeCmd_(ST_STOPPING);
				}
				else {
					executeActingState_(ST_SUSPENDED);
				}
			}
			else if (needParentSynch(stateCurrent_)) {
				setWaitingFor_();
			}
			break;

		case ST_COMPLETE:
			if (abort_) {
				executeCmd_(ST_ABORTING);
			}
			else if (stateComplete_) {
				if (stop_) {
					executeCmd_(ST_STOPPING);
				}
				else if (reset_) {
					executeCmd_(ST_RESETTING);
				}
			}
			else if (stop_ || reset_) {
				setWaitingFor_();
			}
			break;

		case ST_DEACTIVATING:
			if (stateComplete_) {
				executeActingState_(ST_DEACTIVATED);
			}
			else {
				setWaitingFor_();
			}
			break;

		case ST_DEACTIVATED:
			checkActivationCondition_();
			if (stateComplete_) {
				if (activate_) {
					executeCmd_(ST_ACTIVATING);
				}
			}
			else if (activate_) {
				setWaitingFor_();
			}
			break;

		case ST_ACTIVATING:
			if (stateComplete_) {
				executeActingState_(ST_STOPPED);
			}
			else {
				setWaitingFor_();
			}
			break;
	}
}

		// -----------------------------------------------------------------------------

void PackMLModule::checkActivationCondition_()
{

	switch (activationCondition_) {
		case 0:
			activate_ = true;
			break;
		case 1: // by parent: do nothing
			break;
		case 2:
			activate_ = activationPv_;;
			deactivate_ = !activate_;
			break;

		default:
			break;
	}

}

		// -----------------------------------------------------------------------------
```

#### PackMLModuleEnums.hpp
```cpp
#ifndef __PACKMLMODULE_ENUMS_HPP__
#define __PACKMLMODULE_ENUMS_HPP__

enum PackMLModuleStateEnu {
	ST_UNDEFINED = 0,
	ST_CLEARING = 1,
	ST_STOPPED = 2,
	ST_STARTING = 3,
	ST_IDLE = 4,
	ST_SUSPENDED = 5,
	ST_EXECUTE = 6,
	ST_STOPPING = 7,
	ST_ABORTING = 8,
	ST_ABORTED = 9,
	ST_HOLDING = 10,
	ST_HELD = 11,
	ST_UNHOLDING = 12,
	ST_SUSPENDING = 13,
	ST_UNSUSPENDING = 14,
	ST_RESETTING = 15,
	ST_COMPLETING = 16,
	ST_COMPLETE = 17,
	ST_DEACTIVATING = 30,
	ST_DEACTIVATED = 31,
	ST_ACTIVATING = 32
};

enum PackMLModuleEnu {
	NO_ERROR = 0,
	WARNING_INVALID_CMD = 1,
	INFO_PARENT_NOT_ACTIVE = 2,
	ERROR_BLAH = 3,
};

#endif
```

#### PackMLModuleSharedInfo.hpp
```cpp
#ifndef __PACKMLMODULESHAREDINFO_HPP__
#define __PACKMLMODULESHAREDINFO_HPP__

#include "PackMLModuleEnums.hpp"

class PackMLModuleSharedInfo
{
	public:
	// add public members and methods
	PackMLModuleSharedInfo() :
		pName_(nullptr),
		modeCurrent_(0),
		stateCurrent_(ST_UNDEFINED),
		subStateCurrent_(0),
		stateComplete_(false),
		moduleId_(0),
		hierarchyLevel_(0)
	{stateInfo_ = "";}

	const char* getName(){
		if(pName_ == nullptr)
			return "";
		return pName_;
	}

	const char* getStateInfo(){
		return stateInfo_.c_str();
	}

	long int getModeCurrent(){
		return modeCurrent_;
	}

	PackMLModuleStateEnu getStateCurrent(){
		return stateCurrent_;
	}

	long int getSubStateCurrent(){
		return subStateCurrent_;
	}

	bool getStateComplete(){
		return stateComplete_;
	}

	void setValues(const char *pName,
		long int modeCurrent,
		PackMLModuleStateEnu stateCurrent,
		long int subStateCurrent,
		bool stateComplete,
		unsigned short hierarchyLevel,
		unsigned long moduleId,
		const char *pStateInfo)
	{

		if (moduleId_ == 0) {
			moduleId_ = moduleId;
			hierarchyLevel_ = hierarchyLevel;

			pName_ = pName;
			modeCurrent_ = modeCurrent;
			stateCurrent_ = stateCurrent;
			subStateCurrent_ = subStateCurrent;
			stateComplete_ = stateComplete;
			stateInfo_ = pStateInfo;
			return;
		}

		// lets the module overwrite the values anyway
		if (hierarchyLevel_ < hierarchyLevel) {
			moduleId_ = moduleId;
			hierarchyLevel_ = hierarchyLevel;

			pName_ = pName;
			modeCurrent_ = modeCurrent;
			stateCurrent_ = stateCurrent;
			subStateCurrent_ = subStateCurrent;
			stateComplete_ = stateComplete;
			stateInfo_ = pStateInfo;
			return;
		}

		// Relevant for waiting for and blocked/starved
		if (moduleId_ == moduleId) {
			pName_ = pName;
			modeCurrent_ = modeCurrent;
			stateCurrent_ = stateCurrent;
			subStateCurrent_ = subStateCurrent;
			stateComplete_ = stateComplete;
			stateInfo_ = pStateInfo;
		}
	}

	// -----------------------------------------------------------------------------

	void resetValues(unsigned long moduleId)
	{
		if (moduleId_ == moduleId) {
			hierarchyLevel_ = 0;
			moduleId_ = 0;

			pName_ = nullptr;
			modeCurrent_ = 0;
			stateCurrent_ = ST_UNDEFINED;
			subStateCurrent_ = 0;
			stateComplete_ = false;
			stateInfo_ = "";
		}
	}

	unsigned short getHierarchyLevel(){ return hierarchyLevel_; }

	private:

	const char* pName_;
	long int modeCurrent_;
	PackMLModuleStateEnu stateCurrent_;
	long int subStateCurrent_;
	bool stateComplete_;
	std::string stateInfo_;

	unsigned long int moduleId_;
	unsigned short hierarchyLevel_;

};

#endif
```

#### PackMLModuleTable.hpp
```cpp
#ifndef __PACKMLMODULETABLE_HPP__
#define __PACKMLMODULETABLE_HPP__

#include "PackMLModule.hpp"

class PackMLModuleTable
{
	public:
	// add public members and methods
	PackMLModuleTable() : semaphore_(), em_() {

	}

	PackMLModule* getModuleByName(const char* pName){
		unsigned long int moduleId = generateId_(pName);

		if(moduleId == 0)
			return nullptr;

		for(unsigned long int i = 0; i < em_.size(); i++ ){
			if(em_[i]->getModuleId() == moduleId){
				return em_[i];
			}
		}
		return nullptr;
	}

	unsigned long int getModuleIndexByName(const char* pName){
		unsigned long int moduleId = generateId_(pName);

		if(moduleId == 0)
			return 0xFFFFFFFF;

		for(unsigned long int i = 0; i < em_.size(); i++ ){
			if(em_[i]->getModuleId() == moduleId){
				return i;
			}
		}
		return 0xFFFFFFFF;
	}

	PackMLModule* getModuleByIdx(unsigned long int idx){
		return em_[idx % em_.size()];
	}

	bool registerEm(unsigned long int moduleAdr, unsigned long int* moduleIndex = nullptr){

		if(!semaphore_.acquire())
			return false;

		PackMLModule* pPackMLModule = reinterpret_cast<PackMLModule*>(moduleAdr);
		pPackMLModule = getModuleByName(pPackMLModule->getModuleName());

		if(pPackMLModule == nullptr){
			em_.push_back(reinterpret_cast<PackMLModule*>(moduleAdr));

			if(moduleIndex != nullptr){
				*moduleIndex = em_.size() - 1;
			}
		} else {
			if(moduleIndex != nullptr){
				*moduleIndex = getModuleIndexByName(pPackMLModule->getModuleName());
			}
		}

		semaphore_.release();
		return true;
	}

	bool registerEm(PackMLModule* pEm, unsigned long int* moduleIndex = nullptr){

		if(!semaphore_.acquire())
			return false;

		PackMLModule* pPackMLModule = getModuleByName(pEm->getModuleName());

		if(pPackMLModule == nullptr){
			em_.push_back(pEm);

			if(moduleIndex != nullptr){
				*moduleIndex = em_.size() - 1;
			}
		} else {
			if(moduleIndex != nullptr){
				*moduleIndex = getModuleIndexByName(pPackMLModule->getModuleName());
			}
		}

		semaphore_.release();
		return true;
	}

	unsigned long int getNumberOfRoots(){
		unsigned long int rootIdx = 0;

		for(unsigned long int i = 0; i < em_.size(); i++ ){
			if(em_[i]->getHierarchyLevel() == 0){
				rootIdx++;
			}
		}
		return rootIdx;
	}

	unsigned long int getNumberOfModules(){
		return em_.size();
	}

	PackMLModule* getRootModuleByIdx(unsigned long int idx){

		unsigned long int rootIdx = 0;

		for(unsigned long int i = 0; i < em_.size(); i++ ){
			if(em_[i]->getHierarchyLevel() == 0){

				if(rootIdx == idx)
					return em_[i];

				rootIdx++;
			}
		}
		return nullptr;
	}

	private:
	// used during the registration
	AtomicSemaphore semaphore_;
	std::vector<PackMLModule*> em_;

	unsigned long generateId_(const char *pName)
	{
		unsigned long int N = strlen(pName);
		unsigned long int b    = 378551;
		unsigned long int a    = 63689;
		unsigned long int hash = 0;

		for(std::size_t i = 0; i < N; i++)
		{
			hash = hash * a + pName[i];
			a    = a * b;
		}

		return (hash & 0x7FFFFFFF);
	}

};

#endif
```

#### AtomicSemaphore.hpp
```cpp
#ifndef __ATOMIC_SEMAPHORE_HPP__
#define __ATOMIC_SEMAPHORE_HPP__

#include <atomic>

class AtomicSemaphore {
	std::atomic<bool> flag_;
	public:

	bool acquire() {
		return !std::atomic_exchange_explicit(&flag_, true, std::memory_order_acquire);
	}

	void release() {
		std::atomic_store_explicit(&flag_, false, std::memory_order_release);
	}

	bool occupied() {
		return flag_.load();
	}

	AtomicSemaphore(const AtomicSemaphore& source) {
		flag_.store(source.flag_.load());
	}

	AtomicSemaphore& operator=(const AtomicSemaphore& source) {
		flag_.store(source.flag_.load());
		return *this;
	}

	AtomicSemaphore() {
		flag_.store(false);
	}
};

#endif
```

### global.typ
```iecst
(*
Program: Main

Description
(short summary)

*)
(*========== INPUTS ==========*)

TYPE
	MainInputCommandType : 	STRUCT
		Abort : BOOL; (*Go to state Aborting - Can be set in all states except Aborting and Aborted.*)
		Clear : BOOL; (*Go to state Clearing - Can only be set in state Aborted.*)
		Stop : BOOL; (*Go to state Stopping - Can be set in all states except Aborting, Aborted, Clearing, Stopping and Stopped.*)
		Reset : BOOL; (*Go to state Resetting - Can only be set in state Stopped.*)
		Start : BOOL; (*Go to state Starting - Can only be set in state Idle.*)
		Hold : BOOL; (*Go to state Holding. Can only be set in state Execute.*)
		Unhold : BOOL; (*Go to state Unholding. Can only be set in state Held.*)
		Suspend : BOOL; (*Go to state Suspending. Can only be set in state Execute.*)
		Unsuspend : BOOL; (*Go to state Unsuspending. Can only be set in state Suspended.*)
		Complete : BOOL; (*Go to state Completing. Can only be set in state Execute*)
	END_STRUCT;
	MainInputStatusType : 	STRUCT
		SetupComplete : BOOL;
	END_STRUCT;
	MainInputType : 	STRUCT
		Force : BOOL;
		Command : MainInputCommandType;
		Status : MainInputStatusType;
	END_STRUCT;
END_TYPE

(*========== OUTPUTS ==========*)

TYPE
	MainOutputCommandType : 	STRUCT
		NewCommand : BOOL;
	END_STRUCT;
	MainOutputStatusType : 	STRUCT
		NewStatus : BOOL;
	END_STRUCT;
	MainOutputType : 	STRUCT
		Command : MainOutputCommandType;
		Status : MainOutputStatusType;
		Assembly : McAcp6DAsmInfoType;
	END_STRUCT;
END_TYPE

(*========== SETTINGS ==========*)

TYPE
	MainSettingsType : 	STRUCT
		Enable : BOOL;
	END_STRUCT;
END_TYPE

(*========== INTERFACE ==========*)

TYPE
	MainType : 	STRUCT
		Error : GeneralErrorInfoType;
		Input : MainInputType;
		Output : MainOutputType;
		Settings : MainSettingsType;
	END_STRUCT;
END_TYPE
```

### Program Logical/src/Main/Main (IEC)

#### Main.st
```iecst
PROGRAM _INIT

	gCommInput;
	gCommOutput;

    // Access the task interface
	task ACCESS ADR(gMain);

	// Register module config interface for common setup/parametrization functionality
	//fb.MpRecipeRegPar_settings(MpLink := ADR(gSystemSettings), Enable := TRUE , PVName := ADR('gMain.settings'), Category := ADR('Main'));

	// Check for simulator
	//task.IsSimulated := DiagCpuIsSimulated();

	// Calculate home positions for shuttles
	FOR i := 0 TO gMAX_INDEX_SHUTTLE DO
		local.homePosition[i].x := DINT_TO_REAL(420 + (i MOD 2) * 120) / 1000;
		local.homePosition[i].y := DINT_TO_REAL(540 + (i / 2) * 120) / 1000;
	END_FOR;

	// PackML setup
	// =================================================================================================================
	em.Setup.Name := 'Main';
	em.Setup.ParentName := '';

END_PROGRAM

PROGRAM _CYCLIC

    // Access task interface
    // =================================================================================================================
	task ACCESS ADR(gMain);

	// Inputs
	// =================================================================================================================
	IF NOT task.Input.Force THEN

	END_IF

	// Task state machine
	// =================================================================================================================
	// PackML state machine execution
	PackML_state_machine;

	// Detect state change events
	// =================================================================================================================
	// Record information which state caused abort
	fb.R_TRIG_Abort(CLK := em.Command.Abort);

	IF fb.R_TRIG_Abort.Q THEN
		task.Error.State := em.StateCurrent;
		task.Error.SubState := em.SubState;
		task.Error.Description := em.StateInfo;
	END_IF;

	// State change event
	fb.rtStateComplete(CLK := em.Command.StateComplete);

	IF fb.rtStateComplete.Q THEN
		em.StateInfo := '';
		brsmemset(ADR(actions_state), 0, SIZEOF(actions_state));
	END_IF;

	// Substate changed event
	IF em.SubState <> local.lastSubState THEN
		// Reset actions always when state changes
		em.StateInfo := '';
		brsmemset(ADR(actions_substate), 0, SIZEOF(actions_substate));
		local.lastSubState := em.SubState;
	END_IF;

	// Command rising edge detection
	// =================================================================================================================
	commands.Abort(CLK := (task.Input.Command.Abort OR gDI.Button3));
	commands.Clear(CLK := (task.Input.Command.Clear OR gDI.Button3));
	commands.Complete(CLK := task.Input.Command.Complete);
	commands.Hold(CLK := task.Input.Command.Hold);
	commands.Reset(CLK := (task.Input.Command.Reset OR gDI.Button1));
	commands.Start(CLK := (task.Input.Command.Start OR gDI.Button1));
	commands.Stop(CLK := (task.Input.Command.Stop OR gDI.Button2));
	commands.Suspend(CLK := task.Input.Command.Suspend);
	commands.Unhold(CLK := task.Input.Command.Unhold);
	commands.Unsuspend(CLK := task.Input.Command.Unsuspend);

	IF commands.Abort.Q THEN em.Command.Abort := TRUE; END_IF;
	IF commands.Clear.Q THEN em.Command.Clear := TRUE; END_IF;
	IF commands.Complete.Q THEN em.Command.Complete := TRUE; END_IF;
	IF commands.Hold.Q THEN em.Command.Hold := TRUE; END_IF;
	IF commands.Reset.Q THEN em.Command.Reset := TRUE; END_IF;
	IF commands.Start.Q THEN em.Command.Start := TRUE; END_IF;
	IF commands.Stop.Q THEN em.Command.Stop := TRUE; END_IF;
	IF commands.Suspend.Q THEN em.Command.Suspend := TRUE; END_IF;
	IF commands.Unhold.Q THEN em.Command.Unhold := TRUE; END_IF;
	IF commands.Unsuspend.Q THEN em.Command.Unsuspend := TRUE; END_IF;

	// PackML equipment module
	// =================================================================================================================
	em();

	// Function calls
	// =================================================================================================================
	fb.AssemblyReadInfo.Assembly := ADR(gAssembly6D_Big);
	fb.AssemblyReadInfo();

	fb.AssemblyPowerOn.Assembly := ADR(gAssembly6D_Big);
	fb.AssemblyPowerOn.Execute := actions_substate.assemblyPowerOn;
	fb.AssemblyPowerOn();

	fb.AssemblyPowerOff.Assembly := ADR(gAssembly6D_Big);
	fb.AssemblyPowerOff.Execute := actions_substate.assemblyPowerOff;
	fb.AssemblyPowerOff();

	fb.AssemblyReset.Assembly := ADR(gAssembly6D_Big);
	fb.AssemblyReset.Execute := actions_substate.assemblyReset;
	fb.AssemblyReset();

	fb.AssemblyStop.Assembly := ADR(gAssembly6D_Big);
	fb.AssemblyStop.Execute := actions_substate.assemblyStop;
	fb.AssemblyStop();

	fb.WaitUntilAllDone.Execute := actions_substate.waitUntilAllDone;
	fb.WaitUntilAllDone();

	fb.AssemblyReadShIDTable.Assembly := ADR(gAssembly6D_Big);
	fb.AssemblyReadShIDTable.Execute := actions_substate.readShuttleIDs;
	fb.AssemblyReadShIDTable();

	fb.MoveInPlaneAsync.Assembly := ADR(gAssembly6D_Big);
	fb.MoveInPlaneAsync.Execute := actions_substate.homeShuttles;
	fb.MoveInPlaneAsync();

	fb.MoveShortAxis.Execute := actions_substate.moveShortAxis;
	fb.MoveShortAxis();

	fb.AssemblyGetShuttle.Assembly := ADR(gAssembly6D_Big);
	fb.AssemblyGetShuttle.Enable := actions_state.getShuttles;
	fb.AssemblyGetShuttle.Next := actions_substate.getNextShuttle;
	fb.AssemblyGetShuttle();

	// Task output
	// =================================================================================================================
	task.Output.Assembly := fb.AssemblyReadInfo.AssemblyInfo;

	// IO
	// =================================================================================================================
	gDO.Button1_Led := FALSE;
	gDO.Button2_Led := FALSE;
	gDO.Button3_Led := FALSE;

	CASE em.StateCurrent OF
		STATE_ACTIVATING:
//			gDO.Button1_Led := fb.LampSequence.Lamp1;
//			gDO.Button2_Led := fb.LampSequence.Lamp2;
			//			gDO.Button3_Led := fb.LampSequence.Lamp3;
			gDO.Button1_Led := TRUE;
			gDO.Button2_Led := TRUE;
			gDO.Button3_Led := TRUE;

		STATE_EXECUTE:
			gDO.Button1_Led := TRUE;
		STATE_IDLE:
			gDO.Button1_Led := fb.Pulse_slow.Q;
		STATE_STARTING, STATE_RESETTING:
			gDO.Button1_Led := TRUE;

		STATE_STOPPING:
			gDO.Button2_Led := TRUE;
		STATE_STOPPED:
			gDO.Button1_Led := fb.Pulse_slow.Q;
			gDO.Button2_Led := TRUE;

		STATE_ABORTING:
			gDO.Button3_Led := TRUE;
		STATE_ABORTED:
			gDO.Button3_Led := fb.Pulse_slow.Q;
		STATE_CLEARING:
			gDO.Button3_Led := TRUE;
	END_CASE;

	fb.Pulse_slow.T_on := T#500ms;
	fb.Pulse_slow.T_off := T#500ms;
	fb.Pulse_slow(Execute := TRUE);

	// Task diagnostics
	// =================================================================================================================
	gTasks.Main.State := em.StateCurrent;
	gTasks.Main.SubState := em.SubState;
	gTasks.Main.Mode := em.ModeID;
	gTasks.Main.StateComplete := em.Command.StateComplete;
	gTasks.Main.StateInfo := em.StateInfo;
	gTasks.Main.WaitingForTask := em.Info.WaitingFor.Name;
	gTasks.Main.Error := task.Error;

END_PROGRAM

PROGRAM _EXIT

END_PROGRAM
```

#### local.typ
```iecst
TYPE
	MainFbType : 	STRUCT
		MpRecipeRegPar_settings : BOOL;
		AssemblyReadInfo : MC_BR_AsmReadInfo_Acp6D;
		AssemblyPowerOn : MC_BR_AsmPowerOn_Acp6D;
		AssemblyPowerOff : MC_BR_AsmPowerOff_Acp6D;
		AssemblyReset : MC_BR_AsmReset_Acp6D;
		AssemblyGetShuttle : MC_BR_AsmGetShuttle_Acp6D;
		AssemblyStop : MC_BR_AsmStop_Acp6D;
		AssemblyReadShIDTable : MC_BR_AsmReadShIDTable_Acp6D;
		MoveInPlaneAsync : MC_BR_MoveInPlaneAsync_Acp6D;
		WaitUntilAllDone : fdWaitUntilAllDone;
		R_TRIG_Abort : R_TRIG;
		TON_ShuttleScan : TON;
		MoveShortAxis : MC_BR_MoveShortAxis_Acp6D;
		rtStateComplete : R_TRIG;
		Pulse_slow : fdPulse;
	END_STRUCT;
	MainLocalType : 	STRUCT
		lastSubState : DINT;
		shuttleIndex : DINT;
		homePosition : ARRAY[0..gMAX_INDEX_SHUTTLE]OF MainHomePositionType;
		shuttlesCount : USINT;
		lastReadShuttleID : UINT;
	END_STRUCT;
	MainActionsStateType : 	STRUCT
		getShuttles : BOOL; (*Task actions are not automatically reset*)
	END_STRUCT;
	MainActionsSubstateType : 	STRUCT
		assemblyPowerOn : BOOL; (*Task actions are not automatically reset*)
		assemblyPowerOff : BOOL; (*Task actions are not automatically reset*)
		assemblyReset : BOOL; (*Task actions are not automatically reset*)
		assemblyStop : BOOL; (*Task actions are not automatically reset*)
		getNextShuttle : BOOL;
		readShuttleIDs : BOOL; (*Task actions are not automatically reset*)
		homeShuttles : BOOL; (*Task actions are not automatically reset*)
		waitUntilAllDone : BOOL;
		moveShortAxis : BOOL;
	END_STRUCT;
	MainHmiType : 	STRUCT
		isRunning : BOOL;
	END_STRUCT;
	MainHomePositionType : 	STRUCT
		x : REAL;
		y : REAL;
	END_STRUCT;
	MainCommandsType : 	STRUCT
		Abort : R_TRIG; (*Go to state Aborting - Can be set in all states except Aborting and Aborted.*)
		Clear : R_TRIG; (*Go to state Clearing - Can only be set in state Aborted.*)
		Stop : R_TRIG; (*Go to state Stopping - Can be set in all states except Aborting, Aborted, Clearing, Stopping and Stopped.*)
		Reset : R_TRIG; (*Go to state Resetting - Can only be set in state Stopped.*)
		Start : R_TRIG; (*Go to state Starting - Can only be set in state Idle.*)
		Hold : R_TRIG; (*Go to state Holding. Can only be set in state Execute.*)
		Unhold : R_TRIG; (*Go to state Unholding. Can only be set in state Held.*)
		Suspend : R_TRIG; (*Go to state Suspending. Can only be set in state Execute.*)
		Unsuspend : R_TRIG; (*Go to state Unsuspending. Can only be set in state Suspended.*)
		Complete : R_TRIG; (*Go to state Completing. Can only be set in state Execute*)
	END_STRUCT;
END_TYPE
```

#### local.var
```iecst
VAR
	task : REFERENCE TO MainType;
	local : MainLocalType;
	fb : MainFbType;
	hmi : MainHmiType;
	actions_state : MainActionsStateType;
	actions_substate : MainActionsSubstateType;
	commands : MainCommandsType;
	i : DINT;
	x : DINT;
END_VAR
(* ----- PackML ----- *)
VAR
	em : EquipmentModule;
END_VAR
```

#### PackML.st
```iecst
// PackML state machine. Split into different sections that handle
// different logical sequences of PackML stadards' steps
// INFO: Add mode specific code into states by adding CASE structure
// 	CASE em.ModeID OF
//		MODE_PRODUCTION:
//			*CODE*;
//		MODE_MAINTENANCE:
//			*CODE*;
//		MODE_MANUAL:
//			*CODE*;
//		END_CASE
// -----------------------------------------------------------------

ACTION PackML_state_machine:
	// =================================================================================================================
    // Global PackML events
    // =================================================================================================================

    // =================================================================================================================
    // Normal work sequence
    // =================================================================================================================
    CASE em.StateCurrent OF
        STATE_STOPPED:
            em.StateInfo := 'Assembly stopped';
			// -----------------------------------------------------------------
			em.Command.StateComplete := TRUE;

		STATE_RESETTING:
			CASE em.SubState OF
				0:
					em.StateInfo := 'Wait submodules to finish their resets';
					// -----------------------------------------------------------------
					IF gTasks.FastDemo.State = STATE_IDLE THEN
						em.SubState := 10;
					END_IF;
				10:
					em.StateInfo := 'Home all shuttles';
					// -----------------------------------------------------------------
					IF em.Info.OnSubStateEntry THEN
						brsmemset(ADR(fb.MoveInPlaneAsync.Parameters), 0, SIZEOF(fb.MoveInPlaneAsync.Parameters));

						fb.MoveInPlaneAsync.Parameters.Velocity := 1.8;
						fb.MoveInPlaneAsync.Parameters.Acceleration := 15;
						fb.MoveInPlaneAsync.Parameters.Mode := mcACP6D_SHUTTLE_SORTED;
						fb.MoveInPlaneAsync.Parameters.Overhang := FALSE;
						fb.MoveInPlaneAsync.Parameters.MoveOnlySelectedShuttles := FALSE;

						FOR i := 0 TO gShuttles.Count - 1 DO
							fb.MoveInPlaneAsync.Parameters.AsyncPar[i].Shuttle := ADR(gShuttles.Shuttle[i].Ref);
							fb.MoveInPlaneAsync.Parameters.AsyncPar[i].X := local.homePosition[i].x;
							fb.MoveInPlaneAsync.Parameters.AsyncPar[i].Y := local.homePosition[i].y;
						END_FOR;
					END_IF;

					actions_substate.homeShuttles := TRUE;

					IF fb.MoveInPlaneAsync.Done THEN
				 		em.SubState := 20;
					ELSIF fb.MoveInPlaneAsync.Error THEN
						task.Error.Code := fb.MoveInPlaneAsync.ErrorID;
						em.Command.Abort := TRUE;
					END_IF;
				20:
					em.StateInfo := 'Reset short axis orientation of all shuttles';
					// -----------------------------------------------------------------
					IF em.Info.OnSubStateEntry THEN
						fb.MoveShortAxis.Parameters.Mode :=  mcACP6D_MOVE_ABSOLUTE;
						fb.MoveShortAxis.Parameters.Velocity.Rx := 0.1;
						fb.MoveShortAxis.Parameters.Velocity.Ry := 0.1;
						fb.MoveShortAxis.Parameters.Velocity.Rz := 0.1;
						fb.MoveShortAxis.Parameters.Velocity.Z := 0.01;
						fb.MoveShortAxis.Parameters.Position.Rx := 0;
						fb.MoveShortAxis.Parameters.Position.Ry := 0;
						fb.MoveShortAxis.Parameters.Position.Rz := 0;
						fb.MoveShortAxis.Parameters.Position.Z := gDEFAULT_Z;

						local.shuttleIndex := 0;
					END_IF;

					fb.MoveShortAxis.Shuttle := ADR(gShuttles.Shuttle[local.shuttleIndex].Ref);
					actions_substate.moveShortAxis := TRUE;

					IF fb.MoveShortAxis.Acknowledge THEN
						IF local.shuttleIndex < (gShuttles.Count - 1) THEN
							local.shuttleIndex := local.shuttleIndex + 1;
							actions_substate.moveShortAxis := FALSE;
						ELSE
							em.SubState := em.SubState + 1;
						END_IF;
					END_IF;
				21:
					em.StateInfo := 'Wait until all shuttles have completed their moves';
					// -----------------------------------------------------------------
					IF em.Info.OnSubStateEntry THEN
						FOR i := 0 TO MIN(fdMAX_WAIT_SHUTTLE_COUNT, gShuttles.Count) DO
	  						fb.WaitUntilAllDone.Shuttles[i] := gShuttles.Shuttle[i].Ref;
						END_FOR;
					END_IF;

					actions_substate.waitUntilAllDone := TRUE;

					IF fb.WaitUntilAllDone.Done THEN
						em.SubState := 100;
					END_IF;
				100:
					em.StateInfo := 'Done';
					// -----------------------------------------------------------------
					em.Command.StateComplete := TRUE;
			END_CASE;

		STATE_IDLE:
			em.StateInfo := '';
			// -----------------------------------------------------------------
			em.Command.StateComplete := TRUE;

		STATE_STARTING:
			em.StateInfo := '';
			// -----------------------------------------------------------------
			em.Command.StateComplete := TRUE;

		STATE_EXECUTE:
			// -----------------------------------------------------------------
			state_execute;

		STATE_COMPLETING:
			em.StateInfo := '';
			// -----------------------------------------------------------------
			em.Command.StateComplete := TRUE;

		STATE_COMPLETED:
			em.StateInfo := '';
			// -----------------------------------------------------------------
			em.Command.StateComplete := TRUE;

		STATE_STOPPING:
			em.StateInfo := 'Stop assembly';
			// ---------------------------------------------------------------------------------
			actions_substate.assemblyStop := TRUE;

			IF fb.AssemblyStop.Done THEN
				em.Command.StateComplete := TRUE;
			ELSIF fb.AssemblyStop.Error THEN
				task.Error.Code := fb.AssemblyPowerOff.ErrorID;
				em.Command.Abort := TRUE;
			END_IF
	END_CASE

	// =================================================================================================================
	// Module activation sequence
	// =================================================================================================================
	CASE em.StateCurrent OF
		STATE_DEACTIVATING:
			em.StateInfo := '';
			// -----------------------------------------------------------------
			em.Command.StateComplete := TRUE;

		STATE_DEACTIVATED:
			em.StateInfo := '';
			// -----------------------------------------------------------------
			em.Command.StateComplete := TRUE;

		STATE_ACTIVATING:
			// -----------------------------------------------------------------
			sequence_initialize;
	END_CASE

	// =================================================================================================================
	// Abort sequence
	// =================================================================================================================
	CASE em.StateCurrent OF
		STATE_ABORTING:
			em.StateInfo := 'Power off assembly';
			// ---------------------------------------------------------------------------------
			actions_substate.assemblyPowerOff := TRUE;

			IF fb.AssemblyPowerOff.Done THEN
				em.Command.StateComplete := TRUE;
			ELSIF fb.AssemblyPowerOff.Error THEN
				task.Error.Code := fb.AssemblyPowerOff.ErrorID;
				em.Command.StateComplete := TRUE;
			END_IF

		STATE_ABORTED:
			em.StateInfo := 'Assembly powered off';
			// -----------------------------------------------------------------
			em.Command.StateComplete := TRUE;

		STATE_CLEARING:
			// -----------------------------------------------------------------
			sequence_initialize;
	END_CASE

	// =================================================================================================================
	// Hold sequence
	// =================================================================================================================
	CASE em.StateCurrent OF
		STATE_HOLDING:
			em.StateInfo := '';
			// -----------------------------------------------------------------
			em.Command.StateComplete := TRUE;

		STATE_HELD:
			em.StateInfo := '';
			// -----------------------------------------------------------------
			em.Command.StateComplete := TRUE;

		STATE_UNHOLDING:
			em.StateInfo := '';
			// -----------------------------------------------------------------
			em.Command.StateComplete := TRUE;
	END_CASE

	// =================================================================================================================
	// Suspend sequence
	// =================================================================================================================
	CASE em.StateCurrent OF
		STATE_SUSPENDING:
			em.StateInfo := '';
			// -----------------------------------------------------------------
			em.Command.StateComplete := TRUE;

		STATE_SUSPENDED:
			em.StateInfo := '';
			// -----------------------------------------------------------------
			em.Command.StateComplete := TRUE;

        STATE_UNSUSPENDING:
            em.StateInfo := '';
            // -----------------------------------------------------------------
            em.Command.StateComplete := TRUE;

    END_CASE

END_ACTION
```

#### initialize.st
```iecst
ACTION sequence_initialize:
	CASE em.SubState OF
		0:
			em.StateInfo := 'Wait assembly to boot up';
			// ---------------------------------------------------------------------------------
			IF em.Info.OnSubStateEntry THEN
				// Clear old shuttle data
				brsmemset(ADR(gShuttles), 0, SIZEOF(gShuttles));
				brsmemset(ADR(task.Error), 0, SIZEOF(task.Error));
			END_IF;

			fb.AssemblyReadInfo.Enable := TRUE;

			// Wait for the startup phase to be finished
			IF fb.AssemblyReadInfo.Valid THEN
				CASE fb.AssemblyReadInfo.AssemblyInfo.AssemblyState OF
					mcACP6D_ERRORSTOP:
						// Assembly in error state
						em.SubState := 10;
					mcACP6D_STARTUP:
						// Assembly is in the startup phase. Configuration is transferred.
						em.SubState := em.SubState + 1;
					mcACP6D_INVALID_CONFIGURATION:
						// The assembly configuration is invalid. No recovery for this one
					ELSE
						em.SubState := 100;
				END_CASE;
			END_IF

		1:
			em.StateInfo := 'Wait assembly to boot up';
			// ---------------------------------------------------------------------------------
			IF em.Info.OnSubStateEntry THEN
				// Zero the found shuttle count
				local.shuttlesCount := 0;
				fb.TON_ShuttleScan(IN := FALSE);
			END_IF;

			fb.TON_ShuttleScan.PT := T#5s;
			fb.TON_ShuttleScan();

			CASE fb.AssemblyReadInfo.AssemblyInfo.AssemblyState OF
				mcACP6D_STARTUP:
					// Assembly is in the startup phase. Configuration is transferred.
				ELSE
					IF fb.AssemblyReadInfo.AssemblyInfo.CommunicationReady AND (fb.AssemblyReadInfo.AssemblyInfo.Controller6DState <> mcACP6D_STATE_BOOTING) THEN
						// Wait for shuttle scan to finish, reset timer whenevr shuttle count changes
						fb.TON_ShuttleScan.IN := (local.shuttlesCount = fb.AssemblyReadInfo.AssemblyInfo.ShuttlesCount);
						local.shuttlesCount := fb.AssemblyReadInfo.AssemblyInfo.ShuttlesCount;

						IF fb.TON_ShuttleScan.Q THEN
							em.SubState := 0;
						END_IF;
					END_IF;
			END_CASE;
		10:
			em.StateInfo := 'Clear assembly errors';
			// ---------------------------------------------------------------------------------
			actions_substate.assemblyReset := TRUE;

			IF fb.AssemblyReset.Done THEN
				em.SubState := 0;
			ELSIF fb.AssemblyReset.Error THEN
				task.Error.Code := fb.AssemblyReset.ErrorID;
				em.Command.Abort := TRUE;
			END_IF

		100:
			em.StateInfo := 'Assembly power sequence';
			// ---------------------------------------------------------------------------------
			CASE fb.AssemblyReadInfo.AssemblyInfo.AssemblyState OF
				mcACP6D_READY:
					// Assembly powered on -> power off first
					em.SubState := 101;
				mcACP6D_DISABLED:
					// Assembly powered off -> power on
  					em.SubState := 102;
			END_CASE;
		101:
			em.StateInfo := 'Power off assembly';
			// ---------------------------------------------------------------------------------
			actions_substate.assemblyPowerOff := TRUE;

			IF fb.AssemblyPowerOn.Done THEN
				em.SubState := 102;
			ELSIF fb.AssemblyPowerOn.Error THEN
				task.Error.Code := fb.AssemblyPowerOn.ErrorID;
				em.Command.Abort := TRUE;
			END_IF
		102:
			em.StateInfo := 'Power on assembly';
			// ---------------------------------------------------------------------------------
			actions_substate.assemblyPowerOn := TRUE;

			IF fb.AssemblyPowerOn.Done THEN
				em.SubState := 200;
			ELSIF fb.AssemblyPowerOn.Error THEN
				task.Error.Code := fb.AssemblyPowerOn.ErrorID;
				em.Command.Abort := TRUE;
			END_IF

		200:
			em.StateInfo := 'Get all shuttles in the assembly';
			// ---------------------------------------------------------------------------------
			actions_state.getShuttles := TRUE;

			IF fb.AssemblyGetShuttle.Valid THEN
				IF fb.AssemblyGetShuttle.TotalCount > 0 THEN
					em.SubState := em.SubState + 1;
				ELSE
					em.SubState := 210;
				END_IF;
			END_IF
		201:
			em.StateInfo := 'Get all shuttles in the assembly';
			// ---------------------------------------------------------------------------------
			IF em.Info.OnSubStateEntry THEN
				// Clear old shuttle data
				brsmemset(ADR(gShuttles), 0, SIZEOF(gShuttles));
				local.lastReadShuttleID := 0;
			END_IF;

			IF fb.AssemblyGetShuttle.AdditionalInfo.ShuttleID = local.lastReadShuttleID THEN
				actions_substate.getNextShuttle := TRUE;
			ELSE
				gShuttles.Shuttle[gShuttles.Count].ID := fb.AssemblyGetShuttle.AdditionalInfo.ShuttleID;
				gShuttles.Shuttle[gShuttles.Count].Ref := fb.AssemblyGetShuttle.Shuttle;

				local.lastReadShuttleID := fb.AssemblyGetShuttle.AdditionalInfo.ShuttleID;
				gShuttles.Count := gShuttles.Count + 1;
				actions_substate.getNextShuttle := FALSE;
			END_IF;

			// Check if we have found all shuttles or our shuttle list is already full
			IF gShuttles.Count > gMAX_INDEX_SHUTTLE OR fb.AssemblyGetShuttle.RemainingCount = 0 THEN
				em.SubState := 300;
			END_IF;
		210:
			em.StateInfo := 'No shuttles found';
			// ---------------------------------------------------------------------------------

		300:
			em.StateInfo := 'Read shuttle IDs';
			// ---------------------------------------------------------------------------------
			actions_substate.readShuttleIDs := TRUE;

			IF fb.AssemblyReadShIDTable.Done THEN
				FOR i := 0 TO gShuttles.Count - 1 DO
					FOR x := 0 TO gShuttles.Count - 1 DO
						IF fb.AssemblyReadShIDTable.ShIDTable.ShuttleIDs[x] = gShuttles.Shuttle[i].ID THEN
							gShuttles.Shuttle[i].UID.Low := fb.AssemblyReadShIDTable.ShIDTable.UIDLow[x];
							gShuttles.Shuttle[i].UID.High := fb.AssemblyReadShIDTable.ShIDTable.UIDHigh[x];
							EXIT;
						END_IF;
					END_FOR;
				END_FOR;

				em.SubState := 1000;

			ELSIF fb.AssemblyReadShIDTable.Error THEN
				task.Error.Code := fb.AssemblyReadShIDTable.ErrorID;
				em.Command.Abort := TRUE;
			END_IF;

		1000:
			em.StateInfo := 'Done';
			// ---------------------------------------------------------------------------------
			em.Command.StateComplete := TRUE;
	END_CASE;
END_ACTION
```

#### execute.st
```iecst
ACTION state_execute:

	// Start from zero when executing
	IF em.Info.OnStateEntry THEN
		local.shuttleIndex := 0;
	END_IF;

	// No need to wait for anything in this state, all polling is just background process
	em.Command.StateComplete := TRUE;

//	CASE em.SubState OF
//		0:
//			em.StateInfo := 'Update shuttle info';
//			// ---------------------------------------------------------------------------------
//			actions_substate.readShuttleInfo := TRUE;
//
//			fb.ShuttleGetInfo.Shuttle := ADR(gShuttles.Shuttle[local.shuttleIndex].Ref);
//			fb.ShuttleGetInfo.Option := mcACP6D_POSITION_FEEDBACK;
//
//			IF fb.ShuttleGetInfo.Done THEN
//				gShuttles.Shuttle[local.shuttleIndex].State := fb.ShuttleGetInfo.ShuttleInfo.State;
//				gShuttles.Shuttle[local.shuttleIndex].Position := fb.ShuttleGetInfo.ShuttleInfo.Position;
//				gShuttles.Shuttle[local.shuttleIndex].MotionBuffer := fb.ShuttleGetInfo.ShuttleInfo.MotionBuffer;
//				em.SubState := 10;
//			ELSIF fb.ShuttleGetInfo.Error THEN
//				gShuttles.Shuttle[local.shuttleIndex].State := 0;
//				brsmemset(ADR(gShuttles.Shuttle[local.shuttleIndex].Position) ,0 ,SIZEOF(gShuttles.Shuttle[local.shuttleIndex].Position));
//				brsmemset(ADR(gShuttles.Shuttle[local.shuttleIndex].MotionBuffer) ,0 ,SIZEOF(gShuttles.Shuttle[local.shuttleIndex].MotionBuffer));
//				em.SubState := 10;
//			END_IF;
//
//		10:
//			em.StateInfo := 'Get next shuttle';
//			// ---------------------------------------------------------------------------------
//			local.shuttleIndex := local.shuttleIndex + 1;
//			IF local.shuttleIndex > (gShuttles.Count - 1) THEN
//	  			local.shuttleIndex := 0;
//			END_IF;
//
//			em.SubState := 0;
//	END_CASE;
END_ACTION
```

### global.var
```iecst
VAR
	gPower : PowerType := (0);
END_VAR
(**)
VAR CONSTANT
	AUX_POWER_COUNT : USINT := 7;
	AUX_POWER_LAST_INDEX : USINT := AUX_POWER_COUNT-1;
END_VAR
```

### global.typ
```iecst
(*
Program: Power

Description
(short summary)

*)
(*========== STATES ==========*)

TYPE
	PowerStateEnum :
		(
		POWER_INITIALIZE,
		POWER_IDLE,
		POWER_ERROR
		);
END_TYPE

(*========== INPUTS ==========*)

TYPE
	PowerInputCommandType : 	STRUCT
		PowerOn : BOOL;
	END_STRUCT;
	PowerInputType : 	STRUCT
		Force : BOOL;
		Command : PowerInputCommandType;
		SetupComplete : BOOL;
	END_STRUCT;
END_TYPE

(*========== OUTPUTS ==========*)

TYPE
	PowerOutputType : 	STRUCT
		PowerOn : BOOL;
	END_STRUCT;
END_TYPE

(*========== ERRORS ==========*)

TYPE
	PowerErrorType : 	STRUCT
		Active : BOOL;
		Acknowledge : BOOL;
		Code : DINT;
		Description : STRING[80];
	END_STRUCT;
END_TYPE

(*========== INTERFACE ==========*)

TYPE
	AuxPowerUnitType : 	STRUCT
		Command : AuxPowerUnitCommandType;
		CrOk : BOOL;
		OutputEnabled : BOOL;
		StatusRunMode : USINT;
		Current_A : REAL;
		Voltage_V : REAL;
	END_STRUCT;
	AuxPowerUnitCommandType : 	STRUCT
		EnableOutput : BOOL;
		DisableOutput : BOOL;
		AcknowledgeAllErrors : BOOL;
		AcknowledgeAllWarnings : BOOL;
	END_STRUCT;
	PowerType : 	STRUCT
		Error : PowerErrorType;
		Input : PowerInputType;
		Output : PowerOutputType;
		AuxPowerUnit : ARRAY[0..AUX_POWER_LAST_INDEX]OF AuxPowerUnitType;
	END_STRUCT;
END_TYPE
```

### Program Logical/src/Power/Power (IEC)

#### Power.st
```iecst
PROGRAM _INIT

    // Access the task interface
    task ACCESS ADR(gPower);

    // Register module config interface for common setup/parametrization functionality
	//fb.MpRecipeRegPar_settings(MpLink := ADR(gSystemSettings), Enable := TRUE , PVName := ADR('gPower.settings'), Category := ADR('Power'));

	// PackML setup
    // =================================================================================================================
    cm.Setup.Name := 'Power';
	cm.Setup.ParentName := 'Main';

	local.automaticPowerOnAtStart := TRUE;

END_PROGRAM

PROGRAM _CYCLIC

    // Access task interface
    // =================================================================================================================
    task ACCESS ADR(gPower);

    // Inputs
    // =================================================================================================================
    IF NOT task.Input.Force THEN

    END_IF

    // Task state machine
    // =================================================================================================================
    CASE cm.State OF
        0:
            cm.StateInfo := 'Wait for all power units to be ready';
			// ---------------------------------------------------------------------------------
			local.allReadyToStart := TRUE;

			FOR i := 0 TO AUX_POWER_LAST_INDEX DO
				// Check if unit is ready
				IF task.AuxPowerUnit[i].StatusRunMode = 0 OR task.AuxPowerUnit[i].StatusRunMode = 3 THEN
	  				local.allReadyToStart := FALSE;
				END_IF;
			END_FOR;

			IF local.automaticPowerOnAtStart THEN
				task.Input.Command.PowerOn := TRUE;
			END_IF;

			IF local.allReadyToStart THEN
				cm.State := 10;
			END_IF;

		10:
            cm.StateInfo := 'Track power off';
			// ---------------------------------------------------------------------------------
			IF task.Input.Command.PowerOn THEN
				cm.State := 20;
			END_IF;

		20:
			cm.StateInfo := 'Enabling auxiliary power supplies';
			// ---------------------------------------------------------------------------------
			actions.power_on := TRUE;
			IF local.allPowerOn THEN
				cm.State := 30;
			END_IF;

		30:
			cm.StateInfo := 'Track power on';
			// ---------------------------------------------------------------------------------
			IF (NOT task.Input.Command.PowerOn) THEN
				cm.State := 40;
			END_IF;

		40:
			cm.StateInfo := 'Disabling auxiliary power supplies';
			// ---------------------------------------------------------------------------------
			actions.power_off := TRUE;
			IF local.allPowerOff THEN
				cm.State := 10;
			END_IF;
	END_CASE // End of main task logic

	task.Error.Acknowledge := FALSE;

	// Detect state change events
	// =================================================================================================================
	local.onStateEntry := (cm.State <> local.lastState) OR (cm.SubState <> local.lastSubState);

	IF local.onStateEntry THEN
		brsmemset(ADR(actions), 0, SIZEOF(actions));
	END_IF;

	IF cm.State <> local.lastState THEN
		cm.SubState := 0;
		local.lastState := cm.State;
	END_IF

    // Reset current state actions also when substate changes
    IF cm.SubState <> local.lastSubState THEN
        local.lastSubState := cm.SubState;
	END_IF

    // PackML control module
    // =================================================================================================================
	cm();

	// Power command
    // =================================================================================================================
	FOR i := 0 TO AUX_POWER_LAST_INDEX DO
		task.AuxPowerUnit[i].Command.EnableOutput := actions.power_on;
	END_FOR;

	FOR i := 0 TO AUX_POWER_LAST_INDEX DO
		task.AuxPowerUnit[i].Command.DisableOutput := actions.power_off;
	END_FOR;

	// Power on status
	// =================================================================================================================
	local.allPowerOn := TRUE;
	local.allPowerOff := TRUE;

	FOR i := 0 TO AUX_POWER_LAST_INDEX DO
		IF NOT task.AuxPowerUnit[i].OutputEnabled THEN
			local.allPowerOn := FALSE;
		END_IF;

		IF task.AuxPowerUnit[i].OutputEnabled THEN
			local.allPowerOff := FALSE;
		END_IF;
	END_FOR;

	task.Output.PowerOn := local.allPowerOn;

	// Task diagnostics
	// =================================================================================================================
	gTasks.Power.State := cm.State;
	gTasks.Power.SubState := cm.SubState;
	gTasks.Power.StateInfo := cm.StateInfo;

END_PROGRAM

PROGRAM _EXIT

END_PROGRAM
```

#### local.typ
```iecst
TYPE
	PowerFbType : 	STRUCT
		MpRecipeRegPar_settings : BOOL;
	END_STRUCT;
	PowerLocalType : 	STRUCT
		onStateEntry : BOOL;
		lastState : DINT;
		lastSubState : DINT;
		actions : PowerActionsType;
		allReadyToStart : BOOL;
		allPowerOn : BOOL;
		allPowerOff : BOOL;
		automaticPowerOnAtStart : BOOL;
	END_STRUCT;
	PowerActionsType : 	STRUCT
		power_on : BOOL; (*Task actions are not automatically reset*)
		power_off : BOOL; (*Task actions are not automatically reset*)
	END_STRUCT;
	PowerHmiType : 	STRUCT
		isRunning : BOOL;
	END_STRUCT;
END_TYPE
```

#### local.var
```iecst
VAR
	task : REFERENCE TO PowerType;
	local : PowerLocalType;
	fb : PowerFbType;
	hmi : PowerHmiType;
	actions : PowerActionsType;
	i : UDINT;
END_VAR
(* ----- PackML ----- *)
VAR
	cm : ControlModule;
END_VAR
```

### Library Logical/src/FastDemo/FastLib (IEC)

#### Types.typ - Exported data types
```iecst
TYPE
	fdMove6DSyncParametersType : 	STRUCT
		Position : McAcp6DShPositionType;
		Velocity : fdMove6DSyncAllAxesType;
		Acceleration : fdMove6DSyncAllAxesType;
		Mode : McAcp6DMoveModeEnum;
	END_STRUCT;
	fdMove6DSyncAllAxesType : 	STRUCT
		InPlane : REAL;
		Z : REAL;
		Rx : REAL;
		Ry : REAL;
		Rz : REAL;
	END_STRUCT;
	fdMove6DSyncMemberType : 	STRUCT
		DistanceToTarget : fdMove6DSyncAllAxesType;
		TimeToTarget : fdMove6DSyncAllAxesType;
		TimeToEndVelocity : fdMove6DSyncAllAxesType;
		LongestTimeToTarget : REAL;
		TargetVelocity : fdMove6DSyncAllAxesType;
		PositionUpdatePending : BOOL;
	END_STRUCT;
END_TYPE

(**)
(*Stations*)

TYPE
	fdStationParametersType : 	STRUCT
		StationNumber : DINT;
		ShuttleCapacity : UINT;
		CreateVirtualShuttle : BOOL;
		Zone : fdStationParametersZoneType;
		MacroName : STRING[32];
	END_STRUCT;
	fdStationParametersZoneType : 	STRUCT
		Name : STRING[32];
		BottomLeft : McAcp6DInPlaneAxesType;
		TopRight : McAcp6DInPlaneAxesType;
	END_STRUCT;
	fdStationOperationType : 	STRUCT
		Shuttle : MpTrafficShuttleInfoType;
		CommandLabel : fdStationOperationCmdLabelType;
		MoveInPlane : McAcp6DInPlaneParType;
		MoveArc : McAcp6DArcParType;
		Spin : McAcp6DRotaryMotionSpinParType;
		Move6D : McAcp6DMove6DParType;
		MoveShortAxis : McAcp6DShortAxParType;
		WaitCommandLabel : fdStationCmdLbParType;
	END_STRUCT;
	fdStationOperationCmdLabelType : 	STRUCT
		ManualMode : BOOL;
		Label : UINT;
	END_STRUCT;
	fdStationCmdLbParType : 	STRUCT
		TriggerShuttleID : UINT;
		TriggerCmdLb : UINT;
		TriggerType : McAcp6DShWaitCmdLbTriggerEnum;
		LabelType : McAcp6DShWaitCmdLbLabelEnum;
	END_STRUCT;
	fdStationShuttlesType : 	STRUCT
		Count : UINT;
		List : ARRAY[0..fdSTATION_SHUTTLE_LAST_INDEX]OF MpTrafficShuttleInfoType;
	END_STRUCT;
	fdStationCommandsType : 	STRUCT
		AddShuttle : BOOL;
		ErrorReset : BOOL;
		ReleaseAllShuttles : BOOL;
		MoveInPlane : BOOL;
		MoveArc : BOOL;
		MoveShortAxis : BOOL;
		Move6D : BOOL;
		Spin : BOOL;
		SunPlanet : fdStationCommandsSunPlanetType;
		Group : fdStationCommandsGroupType;
		WaitCommandLabel : BOOL;
		WaitUntilAllDone : BOOL;
		MacroRun : BOOL;
		MacroSave : BOOL;
	END_STRUCT;
	fdStationMemberCommandType : 	STRUCT
		Input : fdStationCommandsType;
		GroupCreate : BOOL;
		GroupAddShuttle : BOOL;
		GroupClear : BOOL;
		GroupDelete : BOOL;
		VirtualShuttleCreate : BOOL;
		GetShuttleInfo : BOOL;
		MacroCreate : BOOL;
		MacroDelete : BOOL;
		ZoneCreate : BOOL;
		ZoneGetBarrierInfo : BOOL;
		ZoneFind : BOOL;
	END_STRUCT;
	fdStationMemberStatusType : 	STRUCT
		CommandDone : BOOL;
		CommandAcknowdledge : BOOL;
		CommandError : BOOL;
		ErrorID : DINT;
	END_STRUCT;
	fdStationMemberVarType : 	STRUCT
		SequenceStatePrevious : DINT;
		StateChanged : BOOL;
		ZoneIsEmpty : BOOL;
		Shuttles : fdStationShuttlesType;
		MacroShuttle : MpTrafficShuttleInfoType;
		ShuttleGroup : Mc6DShuttleGroupType;
		ErroredSequenceState : DINT;
		NoCommands : fdStationCommandsType;
		NoCommandActive : BOOL;
		str : STRING[80];
		index : DINT;
		CommandLabel : UINT;
	END_STRUCT;
	fdStationMemberControlType : 	STRUCT
		StationControl : MpTrafficStationControl;
		StationQueueControl : fdStationQueueControl;
		VirtualShuttleCreate : MC_BR_VirtualShCreate_Acp6D;
		GetShuttleInfo : MC_BR_ShGetInfo_Acp6D;
		Enable_EdgeNegative : F_TRIG;
	END_STRUCT;
	fdStationMemberGroupType : 	STRUCT
		Create : MC_BR_ShGroupCreate_Acp6D;
		Clear : MC_BR_ShGroupClear_Acp6D;
		Delete : MC_BR_ShGroupDelete_Acp6D;
		CoupleCtrl : MC_BR_ShGroupCoupleCtrl_Acp6D;
		AddShuttle : MC_BR_ShGroupAddShuttle_Acp6D;
	END_STRUCT;
	fdStationMemberZoneType : 	STRUCT
		Zone : Mc6DZoneType;
		Create : MC_BR_ZoneCreate_Acp6D;
		GetBarrierInfo : MC_BR_ZoneGetBarrierInfo_Acp6D;
		Find : fdFindZone;
	END_STRUCT;
	fdStationMemberMacroType : 	STRUCT
		Create : MC_BR_MacroCreate_Acp6D;
		Delete : MC_BR_MacroDelete_Acp6D;
		Save : MC_BR_MacroSave_Acp6D;
		Run : MC_BR_MacroRun_Acp6D;
	END_STRUCT;
	fdStationMemberMoveType : 	STRUCT
		MoveInPlane : MC_BR_MoveInPlane_Acp6D;
		MoveArc : MC_BR_MoveArc_Acp6D;
		Spin : MC_BR_RotaryMotionSpin_Acp6D;
		Move6D : MC_BR_Move6D_Acp6D;
		MoveShortAxis : MC_BR_MoveShortAxis_Acp6D;
		WaitCommandLabel : MC_BR_ShWaitCmdLb_Acp6D;
		WaitUntilAllDone : fdWaitUntilAllDone;
		SunPlanet : MC_BR_ShPlanet_Acp6D;
	END_STRUCT;
	fdStationCommandsSunPlanetType : 	STRUCT
		Couple : BOOL;
		Decouple : BOOL;
	END_STRUCT;
	fdStationCommandsGroupType : 	STRUCT
		Couple_OwnCenterPoint : BOOL;
		Couple_CommonCenterPoint : BOOL;
		Decouple : BOOL;
	END_STRUCT;
END_TYPE
```

#### Constants.var - Exported constants
```iecst
VAR CONSTANT
	fdMAX_STATION_SHUTTLE_COUNT : DINT := 4;
	fdSTATION_SHUTTLE_LAST_INDEX : DINT := fdMAX_STATION_SHUTTLE_COUNT-1;
	fdMAX_WAIT_SHUTTLE_COUNT : DINT := 35;
END_VAR
```
